# B&R Automation Studio project PLC code - cp (part 2)

### SM_i.ax
```
InitParameter (Version=5.02.1, NcSwId=ACP10)
  ACP10AXIS_typ:
    dig_in:
      level:
        reference = ncACTIV_HI
        pos_hw_end = ncACTIV_HI
        neg_hw_end = ncACTIV_HI
        trigger1 = ncACTIV_HI
        trigger2 = ncACTIV_HI
    encoder_if:
      parameter:
        count_dir = ncINVERSE
        scaling:
          load:
            units = 1000
            rev_motor = 1
    limit:
      parameter:
        v_pos = 10000.0
        v_neg = 10000.0
        a1_pos = 5000.0
        a2_pos = 5000.0
        a1_neg = 5000.0
        a2_neg = 5000.0
        t_jolt = 0.0
        t_in_pos = 0.0
        pos_sw_end = 2000000000
        neg_sw_end = -2000000000
        ds_warning = 100000.0
        ds_stop = 100000.0
        a_stop = 500000.0
        dv_stop = 0.0
        dv_stop_mode = ncOFF
    controller:
      mode = ncPOSITION
      position:
        kv = 50.0
        tn = 0.0
        t_predict = 0.02
        t_total = 0.02
        p_max = 1.0E+30
        i_max = 0.0
      speed:
        kv = 2.0
        tn = 0.0
        t_filter = 0.0
        isq_filter1:
          type = ncOFF
          a0 = 0.0
          a1 = 0.0
          b0 = 0.0
          b1 = 0.0
          b2 = 0.0
          c0_par_id = 0
          c1_par_id = 0
        isq_filter2:
          type = ncOFF
          a0 = 0.0
          a1 = 0.0
          b0 = 0.0
          b1 = 0.0
          b2 = 0.0
          c0_par_id = 0
          c1_par_id = 0
        isq_filter3:
          type = ncOFF
          a0 = 0.0
          a1 = 0.0
          b0 = 0.0
          b1 = 0.0
          b2 = 0.0
          c0_par_id = 0
          c1_par_id = 0
      uf:
        type = ncLINEAR
        auto_config = ncMOTOR_PAR
        u0 = 0.0
        un = 0.0
        fn = 50.0
        k_f_slip = 0.0
      ff:
        torque_load = 0.0
        torque_pos = 0.0
        torque_neg = 0.0
        kv_torque = 0.0
        inertia = 0.0
        t_filter_a = 0.0
    move:
      stop:
        parameter[0]:
          decel_ramp = ncA_LIMIT
          controller = ncON
        parameter[1]:
          decel_ramp = ncA_LIMIT
          controller = ncON
        parameter[2]:
          decel_ramp = ncA_LIMIT
          controller = ncON
        parameter[3]:
          decel_ramp = ncA_LIMIT
          controller = ncON
        quickstop:
          decel_ramp = ncA_LIMIT
          t_jolt = 0
        drive_error:
          decel_ramp = ncA_LIMIT
      homing:
        parameter:
          s = 0
          v_switch = 4000.0
          v_trigger = 4000.0
          a = 2000.0
          mode = ncDIRECT
          edge_sw = ncPOSITIVE
          start_dir = ncPOSITIVE
          trigg_dir = ncPOSITIVE
          ref_pulse = ncOFF
          fix_dir = ncOFF
          tr_s_block = 0.0
          torque_lim = 0.0
          ds_block = 0.0
          ds_stop = 0.0
      basis:
        parameter:
          v_pos = 2000.0
          v_neg = 2000.0
          a1_pos = 1000.0
          a2_pos = 1000.0
          a1_neg = 1000.0
          a2_neg = 1000.0
    message:
      text:
        parameter:
          format = ncBREAK
          columns = 80
          data_modul = acp10etxen
```

### DryerComms.var
```iecst
VAR
	gDryerLocalParams : Dryer_SwParameters; (*Local parameters*)
	gDryerLocalSignals : DryerRemoteData;
END_VAR
```

- RunTextScript.bat (not shown)

### ReadmePrinterConfigurator.txt
```
	From efi Cretaprint Almazora Castellon

(*
View of the machine from the Operator side

>>>>>> LeftHandMachine 					RightHandMachine <<<<<<<<
(BK_A #1 >> BK_B #2)		LOGICAL			(BK_A #2 << BK_B #1)

Vertical:	#2 									Vertical:	#3
IclaNode: 	#5									IclaNode: 	#7
IclaIndex:	#1									IclaIndex:	#2

	          ################-################
	          ################-################
	          ################-################
	          ################-################
	##########################-###########################
	##########################-###########################
	    ######################-#######################
	    ######################-#######################
	    ######################-#######################
	    ######################-#######################

	BLOCK A [1-physical]				BLOCK B [2-physical]

*)
```

### Program Logical/Dryer/Config/Initialize

#### Initialize.st
```iecst
PROGRAM _INIT

	HWInfoCpu.pName := ADR(gDryer.St.HwData.Name);
	HWInfoCpu.first := TRUE;
	HWInfoCpu.enable := TRUE;
	HWInfoCpu();
	gDryer.St.HwData.Family := HWInfoCpu.family;

	// Tranfer permanent vars when PLC is starting
	gMachine.St.HwData.SerialNumber := gPermanentSN;

	gDryer.Pt:= gPermanentDryer;
	gBelt.parSw := gPermanentSwBelt;
	gSimpleBlock[1].parSw := gPermanentSimpleBlock;
	gTransVacuum[1].parSw := gPermanentTrVacuum[1];
	gTransVacuum[2].parSw := gPermanentTrVacuum[2];
	gNirAdphos.Parameters := gPermanentNirAdphos;
	gArcLampGew.Parameters := gPermanentArcLampGew;

	gSimMachine.Parameters.MachineType := gPermanentSimMachinePar.MachineType;

END_PROGRAM

PROGRAM _CYCLIC

	//Assign the ConfigurationID been executed
	projectInfo(Execute:=gDryer.Pt.ConfigNameID=0); //Just to execute if still the configuration has not been read
	IF projectInfo.Done AND NOT projectInfo.Error THEN
		IF brsstrcmp(ADR(GC_CONFIG_DRYER_NOZ2),ADR(projectInfo.ConfigurationID))=0 THEN
			gDryer.Pt.ConfigNameID:=GC_CONFIG_DRYER_NOZ2_ID;
			gSimMachine.Parameters.MachineType := SIM_MACHINE_REAL;
		ELSIF brsstrcmp(ADR(GC_CONFIG_SIMDRYER_NOZ2),ADR(projectInfo.ConfigurationID))=0 THEN
			gDryer.Pt.ConfigNameID:=GC_CONFIG_SIMDRYER_NOZ2_ID;
		ELSE
			gDryer.Pt.ConfigNameID:=0;
		END_IF
		strcpy(ADR(gDryer.Pt.ConfigName),ADR(projectInfo.ConfigurationID));
	END_IF

END_PROGRAM
```

### Program Logical/Dryer/Config/MachineConfigurator

#### AsignCommonData.st
```iecst
ACTION AsignCommonData:

	//Just writing the fixed configuration once per each 5s
	IF NOT (EDGEPOS(gPLC.xBlk_5s) OR gPLC.xFirst_Scan OR xChangedSimMachine) THEN
		RETURN;
	END_IF

	////////////////////////////////////////////////////////////
	/////GENERAL	GENERAL		GENERAL		GENERAL	////////////
	////////////////////////////////////////////////////////////

	gDryer.Pt.CT.rMaxMargin		:= 25.0;
	gDryer.Pt.CT.rMinMargin		:= 5.0;
	gDryer.Pt.CT.rMinThicknessMedia		:= 1.0;
	gDryer.Pt.CT.rMaxThicknessMedia		:= 12.0;
	gDryer.Pt.CT.rDistanceThicknesToPD	:= 187.0;

	/////////////////////////////////////////////////////
	/////BELT	BELT	BELT	BELT	BELT	BELT/////
	/////////////////////////////////////////////////////

	gBelt.parameters.IndexAxis:=1;
	gBelt.parameters.rAcceleration := 1050;
	gBelt.parameters.rSoftDeceleration := 1000;
	gBelt.parameters.rDeceleration := 2200;
	gBelt.parameters.rMaxAcceleration := 1500.0;
	gBelt.parameters.rMaxDeceleration := 2500.0;
	gBelt.parameters.rMaxSpeed := gBelt.states.Hw.rMaxSpeed;

	// From Units measure to meters per minute
	gBelt.parameters.DriveUnit.TransmissionType := TRANS_LINEAL_PERIMETER;
	gBelt.parameters.DriveUnit.LinealPerimeter.PulsesPerTurn := GC_UNITS_BY_REV_DRIVE;
	gBelt.parameters.DriveUnit.LinealPerimeter.GearBox := gBelt.parSw.rGearBox;
	gBelt.parameters.DriveUnit.LinealPerimeter.Perimeter := gBelt.parSw.rAxisLength;

	gBelt.parameters.xExistBelt := TRUE;

	////////////////////////////////////////////////////////////////////////////////////////////////////////////
	// TRANSPORT VACUUM
	////////////////////////////////////////////////////////////////////////////////////////////////////////////
	FOR iIndexTrVacc := 1 TO MAX_LAST_TRANS_VACUUM DO
		gTransVacuum[iIndexTrVacc].Parameters.xInstalled := iIndexTrVacc <= gDryer.Pt.CT.iNumTransVacuum;

		gTransVacuum[iIndexTrVacc].Parameters.parPID.rKp := 0.4;
		gTransVacuum[iIndexTrVacc].Parameters.parPID.rTi := 1.5;
		gTransVacuum[iIndexTrVacc].Parameters.parPID.rKd := 0.0;
		gTransVacuum[iIndexTrVacc].Parameters.parPID.rTd := 0.0;

		gTransVacuum[iIndexTrVacc].Parameters.rMaxSystemVacuum := 18.0;
		gTransVacuum[iIndexTrVacc].Parameters.rMaxSpeed := 3000;
		IF gTransVacuum[iIndexTrVacc].Parameters.rMaxPIDOut = 0 THEN
			gTransVacuum[iIndexTrVacc].Parameters.rMaxPIDOut := 55.0;
		END_IF
	END_FOR
	/////////////////////////////////////////////////////
	/////MODEL	MODEL	MODEL	MODEL	MODEL	MODEL////
	/////////////////////////////////////////////////////

	gThicknessCtrl.parameters.sections[1].xEnabled := TRUE;
	gThicknessCtrl.parameters.iSections := 1;

	gThicknessCtrl.parameters.Detection.ProductDetect.pMediaInProductDetectL1 := gDryer.In.ProductDetect.pPDSignalSensorL1;
	gThicknessCtrl.parameters.Detection.ProductDetect.pMediaInProductDetectL2 := gDryer.In.ProductDetect.pPDSignalSensorL2;

	gThicknessCtrl.parameters.rMountedMediaHeigh := 75.0;

	gThicknessCtrl.parameters.pExtContMedia := ADR(gDryer.Pt.SW.Media);

	// JAM DETECTION DEVICES
	gDryer.Pt.CT.iNumSensorsPerJamDevice := 4;

END_ACTION
```

#### AsignDataDryerNoz2.st
```iecst
ACTION AsignDataDryerNoz2:

	//Just writing the fixed configuration once per each 5s
	IF NOT (EDGEPOS(gPLC.xBlk_5s) OR gPLC.xFirst_Scan OR xChangedSimMachine) THEN
		RETURN;
	END_IF

	////////////////////////////////////////////////////////////
	/////GENERAL	GENERAL		GENERAL		GENERAL	////////////
	////////////////////////////////////////////////////////////
	gDryer.Pt.CT.rMountedMediaLevelInBypassMode	:= 145.0;
	gDryer.Pt.CT.rMaxBeltTorque 		:= 25.0;
	gDryer.Pt.CT.rMaxBeltTempFast 		:= 190.0;
	gDryer.Pt.CT.rMaxBeltTempSlow 		:= 180.0;
	gDryer.Pt.SW.Safety.rMaxBeltSpeedSetPoint := 100.0;
	gDryer.Pt.PDSignalTpe 				:= PDCFG_CARRIAGE;
	gDryer.St.iJamDevices				:= 1;

	gBelt.parameters.xDriveProtectionOK := TRUE; //This machine doesn't have this signal connected to the PLC

	//Here are configured blocks in function of the machine direction
	//When machine is block then we need use correction as block physical 2 because PD is at the same distance than Block 1, for that is change process in function of machine 2 Blcoks or machine 1 block
	gSimpleBlock[1].parameters.iMotorAxisIndex := 2;

	////////////////////////////////////////////////////////////
	/////BLOCK	BLOCK	BLOCK	BLOCK	BLOCK	BLOCK///////////
	////////////////////////////////////////////////////////////
	FOR iIndexBlock:=1 TO gDryer.Pt.CT.iNumBlocks DO

		gSimpleBlock[iIndexBlock].In.xDifferentialOK := TRUE;
		gSimpleBlock[iIndexBlock].In.xDriveProtectionOK := TRUE;
		gSimpleBlock[iIndexBlock].In.xSafetyOK := TRUE;

		gSimpleBlock[iIndexBlock].parameters.Hw.xExistBlock := gDryer.Pt.MachineModel = DryerType_NOZ2_NIR_ARCLAMP;

		gSimpleBlock[iIndexBlock].parSw.xEnableToMovements := TRUE;
		gSimpleBlock[iIndexBlock].parSw.xEnableToPrint := TRUE;

		gSimpleBlock[iIndexBlock].parameters.Motor.rDriveManSpeed		:=10.0;
		gSimpleBlock[iIndexBlock].parameters.Motor.rDriveAutoSpeed		:=30.0;
		gSimpleBlock[iIndexBlock].parameters.Motor.rMinThicknessMedia:= gDryer.Pt.CT.rMinThicknessMedia;
		gSimpleBlock[iIndexBlock].parameters.Motor.rReduceSpeedDistance :=6.0;
		gSimpleBlock[iIndexBlock].parameters.Motor.rAcceleration		:= 172.5;
		gSimpleBlock[iIndexBlock].parameters.Motor.rDeceleration		:= 172.5;

		//Position parameters (mm)
		gSimpleBlock[iIndexBlock].parameters.Motor.rSafePosition	:= 85.0;//Max heigh (theoretically 100)
		gSimpleBlock[iIndexBlock].parameters.Motor.rMinSafePosition	:= 10.0;	//Min heigh
		gSimpleBlock[iIndexBlock].parameters.Motor.rCapPosition		:= 80.0;//CAP

		gSimpleBlock[iIndexBlock].parameters.Motor.DriveUnit.TransmissionType := TRANS_SCREW_PITCH;
		gSimpleBlock[iIndexBlock].parameters.Motor.DriveUnit.ScrewPitch.PulsesPerTurn := GC_UNITS_BY_REV_DRIVE;
		gSimpleBlock[iIndexBlock].parameters.Motor.DriveUnit.ScrewPitch.GearBox := 7.25;
		gSimpleBlock[iIndexBlock].parameters.Motor.DriveUnit.ScrewPitch.Pitch := 5.0;

		gSimpleBlock[iIndexBlock].parameters.Motor.rReferencePosition		:= 20.0;

		//Current Parameters
		gSimpleBlock[iIndexBlock].parameters.Motor.uiMaxCurrentBarsUp		:= 3;
		gSimpleBlock[iIndexBlock].parameters.Motor.uiMaxCurrentBarsDown		:= 1;

		gSimpleBlock[iIndexBlock].parameters.Motor.VerticalDirection:= MOTOR_POSITIVE;

	END_FOR

	///////////////////////////////////////////////////
	/////DING		DING		DING		DING  /////
	///////////////////////////////////////////////////
	gDing.Parameters.xDingInstalled := FALSE;

	///////////////////////////////////////////////////
	//////// DETECTION  DETECTION  DETECTION  /////////
	///////////////////////////////////////////////////

	gBasicDetectMedia.Parameters.xInstalled := TRUE;
	gBasicDetectMedia.Parameters.rCorrection := 12;

	/////////////////////////////////////////////////////
	/////   TRANSPORT_VACUUM  TRANSPORT_VACUUM   ////////
	/////////////////////////////////////////////////////
	gTransVacuum[1].Parameters.xInstalled := TRUE;
	gTransVacuum[1].Parameters.Hw.xSystemWithJoints := FALSE;
	gTransVacuum[1].Parameters.Hw.uiNumBlowers := 2;
	gTransVacuum[1].Parameters.Hw.BlowerData[1].iIndex := 1;
	gTransVacuum[1].Parameters.Hw.BlowerData[1].Direction := MOTOR_NEGATIVE;
	gTransVacuum[1].Parameters.Hw.BlowerData[2].iIndex := 2;
	gTransVacuum[1].Parameters.Hw.BlowerData[2].Direction := MOTOR_NEGATIVE;
	gTransVacuum[1].Parameters.xStartUpEnable := FALSE;
	gAxisInverter[gTransVacuum[1].Parameters.Hw.BlowerData[1].iIndex].Parameters.Hardware.CpuFamily := gDryer.St.HwData.Family;
	gAxisInverter[gTransVacuum[1].Parameters.Hw.BlowerData[2].iIndex].Parameters.Hardware.CpuFamily := gDryer.St.HwData.Family;

	/////////////////////////////////////////////////////
	///// ARCLAMP ARCLAMP ARCLAMP ARCLAMP ARCLAMP ///////
	/////////////////////////////////////////////////////

	gArcLampGew.Parameters.xInstalled := gDryer.Pt.MachineModel = DryerType_NOZ2_NIR_ARCLAMP;

	gArcLampGew.Parameters.CpuFamily := gDryer.St.HwData.Family;
	gArcLampGew.Parameters.iLampQuantity := 2;

	//With real machine, communications cannot be disabled
	IF gDryer.Pt.ConfigNameID <> GC_CONFIG_SIMDRYER_NOZ2_ID THEN
		gArcLampGew.Parameters.xDisableComms := FALSE;
	END_IF

	/////////////////////////////////////////////////////
	///// NIR NIR NIR NIR NIR NIR NIR NIR NIR NIR ///////
	/////////////////////////////////////////////////////
	gNirAdphos.Parameters.xInstalled := gDryer.Pt.MachineModel <> DryerNoType;

	gNirAdphos.Parameters.iTotalModules := 2;
	gNirAdphos.Parameters.CpuFamily := gDryer.St.HwData.Family;
	gNirAdphos.Parameters.rMaxSurfaceTemp := 50;

	gNirAdphos.Parameters.DDC.iLamps := 48;
	gNirAdphos.Parameters.DDC.pIntensityNir1 := ADR(gThicknessCtrl.status.Dry[1].Intensity);
	gNirAdphos.Parameters.DDC.pIntensityNir2 := ADR(gThicknessCtrl.status.Dry[2].Intensity);
	gNirAdphos.Parameters.DDC.rMinIntensityPercentage := 8.0;

	// Thermal inertia configuration
	// Assigning data just if no data to allow setting the data during research
	IF gDryer.Pt.ThermalInertia.iBoardsToStartReducing = 0 THEN
		gDryer.Pt.ThermalInertia.iBoardsToStartReducing := 60;
	END_IF
	IF gDryer.Pt.ThermalInertia.iBoardsToMaxPowerReduction = 0 THEN
		gDryer.Pt.ThermalInertia.iBoardsToMaxPowerReduction := 90;
	END_IF
	IF gDryer.Pt.ThermalInertia.rMaxPowerReduction = 0 THEN
		gDryer.Pt.ThermalInertia.rMaxPowerReduction := 0.85;
	END_IF

	/////////////////////////////////////////////////////
	/////MODEL	MODEL	MODEL	MODEL	MODEL	MODEL////
	/////////////////////////////////////////////////////

	//Configuring machine transport because some values are different in two blocks
	CASE gDryer.Pt.MachineModel OF
		DryerType_NOZ2_NIR,
		DryerType_NOZ2_NIR_ARCLAMP:
			gThicknessCtrl.parameters.iTotalBlocksLengh := 625;
			gThicknessCtrl.parameters.Belt.iDistanceEmptyBeltIni := 685;
	END_CASE;

	gThicknessCtrl.parameters.sections[1].xEnabled	:= TRUE;
	gThicknessCtrl.parameters.sections[1].iStart	:= 1;
	gThicknessCtrl.parameters.sections[1].iEnd		:= 250;

	gThicknessCtrl.parameters.Detection.Basic.xLoadMedia := TRUE;
	gThicknessCtrl.parameters.Detection.Basic.xEnableMediaTracking := TRUE;
	gThicknessCtrl.parameters.Detection.Basic.iMediaFilter := 1; // To avoid adding a 0 in the Tail section

	gThicknessCtrl.parameters.Dry.xEnableMediaTracking := TRUE;

	gThicknessCtrl.parameters.Dry.iLamps := 48;
	gThicknessCtrl.parameters.Dry.rLampOffset := -1435/2;
	gThicknessCtrl.parameters.Dry.rLampWidth := 1435.0/48.0;
	IF gThicknessCtrl.parameters.Dry.rThermalDelay = 0 THEN
		gThicknessCtrl.parameters.Dry.rThermalDelay := 500;
		gThicknessCtrl.parameters.Dry.rCommsDelay := 200;
	END_IF

	gThicknessCtrl.parameters.Dry.Dryers[1].iPosition := 290;
	gThicknessCtrl.parameters.Dry.Dryers[2].iPosition := 415;

	//gThicknessCtrl.parameters.CheckMedia[1].xActive := FALSE; // Deactivated due to sensor reading problems till new sensors will be implemented NOZDRYER-450
	gThicknessCtrl.parameters.CheckMedia[1].CheckPosition := 578;
	gThicknessCtrl.parameters.CheckMedia[1].CheckDelayPosition := 15;
	gThicknessCtrl.parameters.CheckMedia[2].CheckPosition := 578;
	gThicknessCtrl.parameters.CheckMedia[2].CheckDelayPosition := 15;
	gThicknessCtrl.parameters.CheckMedia[2].xActive := gDryer.Pt.SW.xDoubleLine;

	//Jam
	gJamDetect[1].Parameters.iSensorsQuantity := gDryer.Pt.CT.iNumSensorsPerJamDevice;
	gJamDetect[1].Parameters.xJamEnabled	:= TRUE;
	//There are no bars in the dryer, but to use this jam package, designed to be used one jam sensor per bar, we active 4 bars because we have 4 sensors. 2 per NIR module
	gJamDetect[1].Parameters.xBarInstalled[1]:= gNirAdphos.Parameters.xInstalled;
	gJamDetect[1].Parameters.xBarInstalled[2]:= gNirAdphos.Parameters.xInstalled;
	gJamDetect[1].Parameters.xBarInstalled[3]:= gNirAdphos.Parameters.xInstalled;
	gJamDetect[1].Parameters.xBarInstalled[4]:= gNirAdphos.Parameters.xInstalled;
	gJamDetect[1].Parameters.iLowJamCheckDuration[0] := T#1m;
	gJamDetect[1].Parameters.iLowJamTimes[0] := 3;
	gJamDetect[1].Parameters.iLowJamCheckDuration[1] := T#30m;
	gJamDetect[1].Parameters.iLowJamTimes[1] := 10;

END_ACTION
```

#### MachineConfigurator.st
```iecst
PROGRAM _INIT

	//Default values
	gDryerLocalParams.Media.rThickness := 2;
	gDryerLocalParams.Media.rMargin 	:= 10;
	gDryerLocalParams.Media.rLength := 1500;
	gDryerLocalParams.Media.rWidth := 600;

	gThicknessCtrl.parameters.CheckMedia[1].xActive := TRUE;

	//By default, working with comms simulation
	gArcLampGew.Parameters.xDisableComms := TRUE;

END_PROGRAM

PROGRAM _CYCLIC

	//Determine number of last block
	CASE gDryer.Pt.MachineModel OF

		DryerType_NOZ2_NIR,
		DryerType_NOZ2_NIR_ARCLAMP:
			gDryer.Pt.CT.iNumBlocks:=1;
			gDryer.Pt.CT.iNumTransVacuum := 1;
			gDryer.Pt.SW.xMachineDirection := 1; //Machine from left

	END_CASE;

	//Determine machine direction
	// RIGHT: gDryer.Pt.SW.xMachineDirection is 0 or FALSE
	// LEFT:  gDryer.Pt.SW.xMachineDirection is 1 or TRUE
	gDryer.Pt.xLeftHandMachine := gDryer.Pt.SW.xMachineDirection;
	gDryer.Pt.xRightHandMachine:= NOT gDryer.Pt.xLeftHandMachine;

	////////////////////////////////////////////////////////////////////////////////////////////////////////////
	// GENERAL
	////////////////////////////////////////////////////////////////////////////////////////////////////////////

	MachineModel;

	AsignCommonData;

	CASE gDryer.Pt.ConfigNameID OF

		GC_CONFIG_DRYER_NOZ2_ID:
			CASE gDryer.Pt.MachineModel OF
				DryerType_NOZ2_NIR,
				DryerType_NOZ2_NIR_ARCLAMP:
					AsignDataDryerNoz2;
			END_CASE

		GC_CONFIG_SIMDRYER_NOZ2_ID:
			CASE gSimMachine.Parameters.DryerType OF
				SIM_DRYER_NOZ2_NIR,
				SIM_DRYER_NOZ2_NIR_ARCLAMP:
					AsignDataDryerNoz2;
			END_CASE
	END_CASE

	DryerModelCopy := gDryer.Pt.MachineModel;

END_PROGRAM
```

### Program Logical/Dryer/Config/SavePermanent

#### SavePermanent.st
```iecst
PROGRAM _CYCLIC

	// Permanents Vars
	IF brsstrlen(ADR(gDryer.St.HwData.SerialNumber)) > 0 THEN
		gPermanentSN := gDryer.St.HwData.SerialNumber;
	END_IF
	gPermanentDryer:=gDryer.Pt;
	gPermanentSwBelt := gBelt.parSw;
	gPermanentSimpleBlock := gSimpleBlock[1].parSw;
	gPermanentTrVacuum[1] := gTransVacuum[1].parSw;
	gPermanentNirAdphos  := gNirAdphos.Parameters;
	gPermanentArcLampGew  := gArcLampGew.Parameters;

	gPermanentVersion.iVersion0 := gPLC.iVersion0;
	gPermanentVersion.iVersion1 := gPLC.iVersion1;
	gPermanentVersion.iVersion2 := gPLC.iVersion2;
	gPermanentVersion.iVersion3 := gPLC.iVersion3;

	gPermanentSimMachinePar:=gSimMachine.Parameters;

END_PROGRAM
```

### Program Logical/Dryer/DryerCtrl/DryerCtrl_Slow (IEC) - General program

#### Constants.var
```iecst
VAR CONSTANT
	BWMODE_OFF : UINT := 0; (*The blower never is turned on*)
	BWMODE_ON : UINT := 1; (*The blower always is turned on*)
	BWMODE_AUTO : UINT := 2; (*The blower is turned on while moving the belt and a configured time afterwards*)
	SHOT_MIN_TIME_BETWEEN_SHOTS : TIME := T#300MS; (*Minimum time between Printing Shots*)
	BEEP_START_COUNTS : USINT := 7;
END_VAR
```

#### AlarmsSlow.st
```iecst
ACTION AlarmsSlow:

	// Alarm: Platform Incoherence
	gDryer.Al.Alarm.xAlarmPlarformInc:= (gDryer.Pt.MachineModel=DryerNoType) AND NOT gDryer.St.Mode.xZero;

	gDryer.Al.Alarm.xNoActionDangerCollision := FALSE;

	// Warning: Max movemets because bent tile	// Warning: Max movemets because bent tile
	// Warning: Max movemets because bent tile	// Warning: Max movemets because bent tile
	IF EDGEPOS (gDryer.Al.Warning.xBentMedia) THEN
		iBentMediaCounter := iBentMediaCounter + 1;
	END_IF

	//If time without any change, decrease the count of movements
	tonDecreaseMovCount.IN := NOT gDryer.Al.Warning.xMaxMovsBentTile AND NOT gDryer.Al.Warning.xBentMedia AND NOT tonDecreaseMovCount.Q ;
	tonDecreaseMovCount.PT := T#5m;
	tonDecreaseMovCount();
	IF tonDecreaseMovCount.Q THEN
		//Safety decrease to avoid overflow
		iBentMediaCounter:= UINT_SUB(iBentMediaCounter,1);
	END_IF
	IF EDGEPOS(gDryer.Al.Warning.xMaxMovsBentTile) THEN
		iBentMediaCounter:= 0;
	END_IF

	IF 	iBentMediaCounter >= gc_diNumMaxManiobrasPDoblada THEN
		gDryer.Al.Warning.xMaxMovsBentTile:=TRUE;
	ELSIF  gDryer.AutoCmd.xReset THEN
		gDryer.Al.Warning.xMaxMovsBentTile:=FALSE;
	END_IF

	// Raising alarm of stopped media inside.
	// this is a simple way to reset the alarm. A more proper way to remove the alarm would be to
	// use a distanceVar in Thickness_Pos, but this is quite resource consuming, so this would be delayed
	IF gThicknessCtrl.status.MediaPosition.xMediaInside AND EDGENEG(gBelt.states.xRuningBelt) THEN
		gDryer.Al.Warning.xMediaStoppedInside := TRUE;
	ELSIF gThicknessCtrl.status.Belt.xBeltEmpty THEN
		gDryer.Al.Warning.xMediaStoppedInside := FALSE;
	END_IF

	//Sensors errors
	IF gDryer.In.Temp.xBeltSensorError THEN
		gDryer.Al.Warning.xBeltSensorError := TRUE;
	END_IF

	IF gDryer.In.Temp.xBoardInSensorError THEN
		gDryer.Al.Warning.xBoardInSensorError := TRUE;
	END_IF

	IF gDryer.In.Temp.xBoardOutSensorError THEN
		gDryer.Al.Warning.xBoardOutSensorError := TRUE;
	END_IF

	IF gDryer.In.Temp.xAirBlowerInputSensorError THEN
		gDryer.Al.Warning.xAirBlowerInputSensorError := TRUE;
	END_IF

	IF gDryer.In.Temp.xAirBlowerInputSensorError THEN
		gDryer.Al.Warning.xAirBlowerOutputSensorError := TRUE;
	END_IF

	//BELT ALARMS
	tonBeltOvertorque.IN := gBelt.states.rCurrentTorque > gDryer.Pt.CT.rMaxBeltTorque;
	tonBeltOvertorque.PT := t#120s;
	tonBeltOvertorque();
	IF tonBeltOvertorque.Q THEN
		gDryer.Al.Alarm.xAlrBeltOvertorque := TRUE;
	END_IF

	tonBeltOverTempFast.IN := gDryer.St.Temp.rBelt > gDryer.Pt.CT.rMaxBeltTempFast;
	tonBeltOverTempFast.PT := t#2s;
	tonBeltOverTempFast();
	IF tonBeltOverTempFast.Q THEN
		gDryer.Al.Alarm.xAlrBeltOverTempFast := TRUE;
	END_IF

	tonBeltOverTempSlow.IN := gDryer.St.Temp.rBelt > gDryer.Pt.CT.rMaxBeltTempSlow;
	tonBeltOverTempSlow.PT := t#30s;
	tonBeltOverTempSlow();
	IF tonBeltOverTempSlow.Q THEN
		gDryer.Al.Alarm.xAlrBeltOverTempSlow := TRUE;
	END_IF

	IF gJamDetect[1].Alarms.xAlrJamLowCrash THEN
		gDryer.Al.Warning.xJamLowCrash := TRUE;
	END_IF

	PsycallConfChecking;

END_ACTION

ACTION PsycallConfChecking:
	CASE gDryer.Pt.ConfigNameID OF
		GC_CONFIG_DRYER_NOZ2_ID:
			CASE gDryer.Pt.MachineModel OF
				DryerType_NOZ2_NIR,
				DryerType_NOZ2_NIR_ARCLAMP:
					plcCardsOK.0 := NOT X20DIF371_201.ModuleOk;
					plcCardsOK.1 := NOT X20DIF371_202.ModuleOk;
					plcCardsOK.2 := NOT X20DIF371_203.ModuleOk;
					//plcCardsOK.3 := NOT X20PS3300_204.ModuleOk;
					plcCardsOK.4 := NOT X20DOF322_205.ModuleOk;
					plcCardsOK.5 := NOT X20DOF322_206.ModuleOk;
					plcCardsOK.6 := NOT X20AI8321_207.ModuleOk;
					plcCardsOK.7 := NOT X20AO4622_208.ModuleOk;
					plcCardsOK.8 := NOT X20AT4222_209.ModuleOk;
					gDryer.Al.Alarm.xAlrWrongPhysConf := plcCardsOK>0;

				ELSE
					gDryer.Al.Alarm.xAlrWrongPhysConf := TRUE;
			END_CASE

		GC_CONFIG_SIMDRYER_NOZ2_ID:
			gDryer.Al.Alarm.xAlrWrongPhysConf := FALSE;

		ELSE

			gDryer.Al.Alarm.xAlrWrongPhysConf := TRUE;

	END_CASE

END_ACTION
```

#### CleanBelt.st
```iecst
ACTION CleanBelt:

	///////////////////////////////////////////////////////////////////////////////////////////////////////////////////
	// General conditions to clean belt	when machine is in AUTOMATIC OR MANUAL MODES
	///////////////////////////////////////////////////////////////////////////////////////////////////////////////////

	//Cleaning Belt by time. When cleaning, the time is reseted
	tonCleaningByTime.IN:= gBelt.states.xRuningBelt AND gDryer.Pt.SW.CleanBelt.xCleanBeltByTime AND NOT tonCleaningByTime.Q AND NOT xCleanBeltOrder;
	tonCleaningByTime.PT := MAX(tiCleaningBeltByTime, MIN_TIME_FOR_CLEANING_BELT); // Time converted from minutes to miliseconds
	tonCleaningByTime();

	//If the belt is not running, it is not possible to clean it
	IF NOT gBelt.states.xRuningBelt THEN
		RETURN;
	END_IF

	// Tiles counter
	IF gDryer.Pt.SW.CleanBelt.xCleanBeltByTiles AND (EDGEPOS (gDryer.St.xProductDetectL1) OR EDGEPOS(gDryer.St.xProductDetectL2)) THEN
		gDryer.Lg.iTilesCounterToClean:= gDryer.Lg.iTilesCounterToClean+1;
	END_IF

	//Cleaning by tiles. When cleaning, number of tiles is reseted
	IF gDryer.Pt.SW.CleanBelt.xCleanBeltByTiles AND (gDryer.Lg.iTilesCounterToClean >= INT_TO_UINT(iSPTilesToCleanBelt)) THEN
		xCleaningBeltByTiles:= TRUE;
	END_IF

	// Force cleaning applying delay. Why clean continuous is same that condition than force clean?
	IF gDryer.Pt.SW.CleanBelt.xCleanBeltForced THEN
		xCleanBeltForced:= TRUE;
		gDryer.Pt.SW.CleanBelt.xCleanBeltForced := FALSE;
	END_IF

	IF tonCleaningByTime.Q THEN
		xCleaningBeltByTime:=TRUE;
	END_IF

	IF xCleaningBeltByTiles OR xCleaningBeltByTime OR xCleanBeltForced OR gDryer.Pt.SW.CleanBelt.xCleanBeltContinue THEN
		xCleanBeltOrder:=TRUE;

		//Removed orders when cleaning
		xCleaningBeltByTiles:=FALSE;
		gDryer.Lg.iTilesCounterToClean:=0;
		xCleaningBeltByTime:=FALSE;
		xCleanBeltForced := FALSE;

	END_IF

	// Managing the duration of the belt cleaning
	tonCleaningBelt.IN:= xCleanBeltOrder;
	tonCleaningBelt.PT := MAX(gDryer.Pt.SW.CleanBelt.tiCleaningBeltDuration, MIN_DURATION_CLEANING_BELT);
	tonCleaningBelt();

	IF (tonCleaningBelt.Q AND NOT(gDryer.Pt.SW.CleanBelt.xCleanBeltContinue)) OR EDGENEG(gDryer.Pt.SW.CleanBelt.xCleanBeltContinue) THEN
		xCleanBeltOrder:=FALSE;
	END_IF

END_ACTION
```

#### GeneralMachineData.st
```iecst
ACTION GeneralMachineData:

	//////////////////////////////////////////////////////////////////////////////////////////////////////////////////////
	// BELT PARAMS      BELT PARAMS      BELT PARAMS      BELT PARAMS      BELT PARAMS      BELT PARAMS      BELT PARAMS
	// BELT PARAMS      BELT PARAMS      BELT PARAMS      BELT PARAMS      BELT PARAMS      BELT PARAMS      BELT PARAMS
	//////////////////////////////////////////////////////////////////////////////////////////////////////////////////////

	// Cleaning Belt limits cannot be lower than 1
	// Cleaning Belt parameters. Clean Belt disabled/enabled after delay
	tiCleaningBeltByTime	:= MINUTES_TO_TIME(gDryer.Pt.SW.CleanBelt.iCleaningBeltByTime);
	iSPTilesToCleanBelt		:= MAX (gDryer.Pt.SW.CleanBelt.iSPTilesToCleanBelt, MIN_TILES_FOR_CLEANING_BELT);

	////////// Belt Limits //////////////////////////////////
	//[RGP] Sending speed setpoint to gBelt. Not assigned directly from SW so maybe in the future SpeedSetpoint need to be used outside BeltPackage/BeltManager.
	//As done in previous lines by limiting maximum belt speed. //Not been able to have a Zero value in the SetPointSpeed
	gBelt.parameters.rSetPointSpeed := LIMIT(5.0, gDryer.Pt.SW.rBeltSpeedSetPoint, gDryer.Pt.SW.Safety.rMaxBeltSpeedSetPoint);

	// It gets belt direction following if machine configuration is left or right
	gBelt.parameters.Direction:= NOT gDryer.Pt.SW.xMachineDirection;

	////////////////////////////////////////////////////////////////////////////////////////////////////////////
	// MODEL
	////////////////////////////////////////////////////////////////////////////////////////////////////////////

	// Jetting Gap limits
	gDryer.Pt.SW.Media.rMargin:= LIMIT(gDryer.Pt.CT.rMinMargin,gDryer.Pt.SW.Media.rMargin,gDryer.Pt.CT.rMaxMargin);

	// Piece Tickness
	gDryer.Pt.SW.Media.rThickness:= LIMIT(gDryer.Pt.CT.rMinThicknessMedia,gDryer.Pt.SW.Media.rThickness,gDryer.Pt.CT.rMaxThicknessMedia);

	// Counters of shots printed by PD or by simulation
	//Counting out of any FOR. Makes no sense
	IF EDGEPOS (gDryer.St.xProductDetectL1) THEN
		gDryer.Lg.udiPiecesCounterL1:= gDryer.Lg.udiPiecesCounterL1+1;
	END_IF

	IF EDGEPOS (gDryer.St.xProductDetectL2) THEN
		gDryer.Lg.udiPiecesCounterL2:= gDryer.Lg.udiPiecesCounterL2+1;
	END_IF

	// Machine conversions
	gDryer.Lg.udiDifCounters:=0;

END_ACTION
```

#### SoundBeacon.st
```iecst
ACTION SoundBeacon:
	// Acoustic advise
	//
	// AutoReseteable Alarms sound management
	arFanBreakers		(xAlarm:= gDryer.Al.Alarm.xFanBreakers, xSilence:=gDryer.AutoCmd.xMuteAlarms);
	arFan24Vdc			(xAlarm:= gDryer.Al.Alarm.xFan24Vdc, xSilence:=gDryer.AutoCmd.xMuteAlarms);
	arMain24Vdc			(xAlarm:= gDryer.Al.Alarm.xMain24Vdc, xSilence:=gDryer.AutoCmd.xMuteAlarms);
	arBentMedia			(xAlarm:= gDryer.Al.Warning.xBentMedia, xSilence:=gDryer.AutoCmd.xMuteAlarms);
	arPDSensorErrorL1	(xAlarm:= gDryer.Al.Alarm.xPDBrokenSensorL1, xSilence:=gDryer.AutoCmd.xMuteAlarms);
	arPDSensorErrorL2	(xAlarm:= gDryer.Al.Alarm.xPDBrokenSensorL2, xSilence:=gDryer.AutoCmd.xMuteAlarms);
	arWrongPhysConf		(xAlarm:= gDryer.Al.Alarm.xAlrWrongPhysConf, xSilence:=gDryer.AutoCmd.xMuteAlarms);
	arAnyJam			(xAlarm:= gDryer.Al.Alarm.xAlrJam, xSilence:=gDryer.AutoCmd.xMuteAlarms);

	//arAnyStopAlarmMuted	(xAlarm:= gDryer.AlSummary.xAnyAlarm AND gDryer.St.StateMode<>PRINTERGEN_ZERO, xSilence:= gDryer.AutoCmd.xMuteAlarms);

	reasonSoundGen.1 := arFanBreakers.xAlarmSound;
	reasonSoundGen.2 := arFan24Vdc.xAlarmSound;
	reasonSoundGen.3 := arMain24Vdc.xAlarmSound;
	reasonSoundGen.4 := arBentMedia.xAlarmSound;
	reasonSoundGen.5 := arAnyStopAlarmMuted.xAlarmSound;
	reasonSoundGen.6 := arPDSensorErrorL1.xAlarmSound;
	reasonSoundGen.7 := arPDSensorErrorL2.xAlarmSound;
	reasonSoundGen.8 := arWrongPhysConf.xAlarmSound;
	reasonSoundGen.9 := arAnyJam.xAlarmSound;
	reasonSoundGen.25 := gBasicDetectMedia.AlSummary.xAlarmSound;
	reasonSoundGen.26 := gBelt.AlSummary.xAlarmSound;
	reasonSoundGen.27 := gSimpleBlock[1].AlSummary.xAlarmSound;
	reasonSoundGen.28 := gTransVacuum[1].AlSummary.xAlarmSound;
	reasonSoundGen.29 := gNirAdphos.AlSummary.xAlarmSound;
	reasonSoundGen.30 := gArcLampGew.AlSummary.xAlarmSound;
	reasonSoundGen.31 := gThicknessCtrl.Alarms.CheckMedia[1] OR gThicknessCtrl.Alarms.CheckMedia[2];

	gDryer.Al.xAlarmSound:= reasonSoundGen > 0;

	// Alarm sound output
	IF 	gDryer.AutoCmd.xMuteAlarms OR gDryer.In.Buttons.xZero THEN
		gDryer.AlSummary.xAlarmSound:=FALSE;
	ELSE
		gDryer.AlSummary.xAlarmSound:= gDryer.Al.xAlarmSound;
	END_IF;

	SoundAtStart;

	reasonBuzzer.0 := gDryer.AlSummary.xAlarmSound AND (iCountStartSound >= BEEP_START_COUNTS);
	reasonBuzzer.1 := gBelt.states.State = BELT_PREPARING_START  AND gPLC.xBlk_500ms;
	reasonBuzzer.2 := xStartSound;

	gDryer.Out.xBuzzer :=  reasonBuzzer > 0;

END_ACTION

ACTION SoundAtStart:

	//Whit 5, we have 3 beeps at the begining
	IF iCountStartSound >= BEEP_START_COUNTS THEN
		RETURN;
	END_IF

	tonStartSound.IN := NOT tonStartSound.Q;
	tonStartSound.PT := t#1s;
	tonStartSound();

	IF EDGEPOS(tonStartSound.Q) THEN
		iCountStartSound := iCountStartSound + 1;
	END_IF

	xStartSound := (iCountStartSound MOD 2) = 0;

END_ACTION
```

### Program Logical/Dryer/DryerCtrl/DryerCtrl_Fast (IEC) - Machine program

#### DryerCtrl_Fast.var
```iecst
VAR
	xRunBeltNormal : BOOL;
	xRunBeltLab : BOOL;
	xStopBeltWhileCleaning : BOOL;
	xSignalsStopBeltAuto : BOOL;
	xUserRaisesBlocks : BOOL;
	xOrdersRunBeltProduction : BOOL;
	xRunBeltByPass : BOOL;
	xAlarmsStopBeltRun : BOOL;
	enPrinterState : enumEFI_GenMachineState := PRINTERGEN_MANUAL; (*PRINTERGEN_ZERO*)
	enPrinterStatesInAuto : enumEFI_MachineState := PRINTERGEN_ZERO; (*PRINTERGEN_ZERO*)
	rsRunBeltOrderManual : RS;
	srPauseMachine : {REDUND_UNREPLICABLE} RS;
	stDryerAlarmsSummaryReseted : stEFI_AlarmSummary; (*stDingAlarmsReseted : stPhotoCellsAlarms;*)
	stDryerAlarmsReseted : Dryer_Alarms;
	tonStartButton : TON;
	ton_ZeroMode : TON;
	tpAlrBentMedia : TP;
	iIndexBlock : USINT;
	iReasonOut : UDINT;
	iReasonStopGen : UDINT;
	iReasonCritical : UDINT;
	stEventLogState : EventLog_typ;
	stEventLogOutAuto : EventLog_typ;
	stEventLog : EventLog_typ;
	stEventLogStopDrying : EventLog_typ;
	stEventLogCritical : EventLog_typ;
	g_xRunBeltOrderManual : BOOL; (*Belt order in manual filtered*)
	g_xRunBeltOrderAuto : BOOL; (*Belt order in auto*)
	reasonAnyWarningGen : UDINT;
	xEnabledAlarmPDSensor1 : BOOL;
	xEnabledAlarmPDSensor2 : BOOL;
	usiIndex : USINT;
	trgMountedTile : RF_TRIG;
	AutoLocationPrevious : MachineAutoLocation_enum;
	AutoLocationReseted : MachineAutoLocation_enum := MACHLOC_UNDEFINED;
	DryerCommandsReseted : {REDUND_UNREPLICABLE} Dryer_commands_Auto; (*Local parameters*)
	DryerSignalsAuto : REFERENCE TO DryerRemoteData; (*Local parameters*)
	DryerParams : REFERENCE TO Dryer_SwParameters; (*Local parameters*)
	iLastReasonStop : USINT;
	iReasonStop : USINT;
	iReasonSetPause : USINT;
	iReasonResetPause : USINT;
	DryerStatus : DryerMachineStatus_enum;
	DryerStatus_copy : DryerMachineStatus_enum;
	iReasonReadyToDry : USINT;
	xStartedAutoMan : BOOL;
	InputsSwReseted : Dryer_Inputs_Sw;
	tonMovingBeltAfterStop : TON;
END_VAR
VAR CONSTANT
	iHistoryLines : USINT := 25;
END_VAR
VAR
	StateHistory : ARRAY[0..iHistoryLines] OF DryerMachineStatus_enum;
	iIndexHistory : USINT;
	xNirReady : BOOL;
	xArcLampReady : BOOL;
	xAllDryersReady : BOOL;
	xNirStopped : BOOL;
	xArcLampStopped : BOOL;
	xAllDryersStopped : BOOL;
	xNirDrying : BOOL;
	xArcLampDrying : BOOL;
	xAllDryersDrying : BOOL;
	xChangeState : BOOL;
	iReasonSafetyEStop : UINT;
	tonStop : TON;
	xAnyDeviceEnabled : BOOL;
	iReasonJam : UINT;
	iReasonNotEnterAuto : UINT;
	xEdgeStop : BOOL;
	xOrderToCapReceived : BOOL;
	xOrderToPrintReceived : BOOL;
	iReasonCap : UINT;
	iReasonPrint : UINT;
	lastReasonCap : UINT;
	iBlockExecutionsOrder : UDINT;
	lastReasonPrint : UINT;
	iBlockDelay : UDINT;
	gDryerLocalSignalsReseted : DryerRemoteData;
	iReasonStopDrying : UINT;
	tonPreparingEmptyBelt : TON;
	iReasonKeepBlowersOn : UINT;
	xKeepBlowersOn : BOOL; (*To keep blowers running due to certain conditions*)
	xPDCarriageSignalL1 : REFERENCE TO BOOL; (*Use just in MachineInputs*)
	xPDCarriageSignalL2 : REFERENCE TO BOOL; (*Use just in MachineInputs*)
	ton_EmptyBelt : TON;
END_VAR
```

#### Alarms.st
```iecst
ACTION Alarms:

	// SAFETY
	IF NOT gDryer.In.Safety.xEStopFrontOK THEN gDryer.Al.Alarm.Safety.xEStopFront := TRUE; END_IF
	IF NOT gDryer.In.Safety.xEStopRearOK THEN gDryer.Al.Alarm.Safety.xEStopRear := TRUE; END_IF
	//IF NOT gDryer.In.Safety.xRemoteEStopOK THEN gDryer.Al.Alarm.Safety.xRemoteEStop := TRUE; END_IF  //TODO: Remove when working

	IF NOT gDryer.In.Safety.xMovementsEnabled THEN gDryer.Al.Warning.xNotEnabledMovement := TRUE; END_IF

	IF NOT gDryer.In.Safety.xClosedFrontInput OR NOT gDryer.In.Safety.xClosedFrontOutput THEN
		gDryer.Al.Warning.xFrontDoorOpened := TRUE;
	END_IF
	IF NOT gDryer.In.Safety.xClosedRearInput OR NOT gDryer.In.Safety.xClosedRearOutput THEN
		gDryer.Al.Warning.xRearDoorOpened := TRUE;
	END_IF

	iReasonSafetyEStop.0 := gDryer.Al.Alarm.Safety.xEStopFront;
	iReasonSafetyEStop.1 := gDryer.Al.Alarm.Safety.xEStopRear;
	iReasonSafetyEStop.2 := gDryer.Al.Alarm.Safety.xRemoteEStop;
	gDryer.Al.xAlrSafetySystemEStop := iReasonSafetyEStop>0;

	// Warning Alarm raised when a new BentTile is detected. The signal is kept for 5s
	tpAlrBentMedia.IN:=(gDryer.St.AutoMode.xProdORLab) AND EDGEPOS(gThicknessCtrl.status.Heigh.xIncreasedHeigh[1]);
	tpAlrBentMedia.PT:= T#5S;
	tpAlrBentMedia();
	gDryer.Al.Warning.xBentMedia:=tpAlrBentMedia.Q;

	//Count all the increase of heigh of the blocks as bent media
	IF EDGEPOS (tpAlrBentMedia.IN) THEN
		gDryer.Lg.udiBentTilesCounter:= gDryer.Lg.udiBentTilesCounter+1;
	END_IF

	//24VDC Power Supply for IDS
	IF NOT gDryer.In.xMain24VdcOK THEN gDryer.Al.Alarm.xMain24Vdc := TRUE; END_IF
	IF NOT gDryer.In.xFan24VdcOK THEN gDryer.Al.Alarm.xFan24Vdc := TRUE; END_IF
	IF NOT gDryer.In.xFanBreakersOK THEN gDryer.Al.Alarm.xFanBreakers := TRUE; END_IF
	IF gDryer.In.xFanBreakersWarning THEN gDryer.Al.Warning.xFanBreakersHighLoad := TRUE; END_IF

	// Alarm: xUpNotConsent
	gDryer.Al.Alarm.xUpNotConsent:= gDryer.St.AutoMode.xProduction AND
									NOT gDryer.St.xConsent;

	//Alarm: Mounted Piece Inide the Machine
	gDryer.Al.Alarm.xAlarmMountedMedia := gBasicDetectMedia.Alarms.xMountedMedia;
	gDryer.Al.Warning.xMountedMediaInside := gThicknessCtrl.status.MediaPosition.xMountedMediaInside;

	//Jam alarms
	iReasonJam.0 := gJamDetect[1].AlSummary.xAlarmStop;
	iReasonJam.1 := gArcLampGew.Alarms.xJam;
	iReasonJam.2 := gNirAdphos.Alarms.xAnyJam;
	iReasonJam.3 := gJamDetect[1].Alarms.xAlrJamCrash[1];
	iReasonJam.4 := gJamDetect[1].Alarms.xAlrJamCrash[2];
	iReasonJam.5 := gJamDetect[1].Alarms.xAlrJamCrash[3];
	iReasonJam.6 := gJamDetect[1].Alarms.xAlrJamCrash[4];
	//iReasonJam.7 := gThicknessCtrl.Alarms.CheckMedia[1] OR gThicknessCtrl.Alarms.CheckMedia[2];
	IF iReasonJam>0 THEN
		gDryer.Al.Alarm.xAlrJam := TRUE;
	END_IF

	IF gDryer.In.xOpenDoorsKey THEN
		gDryer.Al.Warning.xKeyMantenanceActive := TRUE;
	END_IF

	//Alarm: Broken PD
	CalcPDSensorAlarm;

END_ACTION

ACTION CalcPDSensorAlarm:

	//When no sensor is connected, cannot be checked
	IF (gDryer.Pt.PDSignalTpe <> PDCFG_SENSOR AND gDryer.Pt.PDSignalTpe <> PDCFG_SENSOR_AND_CARRIAGE) THEN
		gDryer.Lg.udiPiecesCounterErrorL1 := 0;
		gDryer.Lg.udiPiecesCounterErrorL2 := 0;
		RETURN;
	END_IF

	//Reset counter when belt is stoped or not in printin
	IF NOT gBelt.states.xRuningBelt OR NOT gDryer.St.Position.xInPrint THEN
		gDryer.Lg.udiPiecesCounterErrorL1 := 0;
		gDryer.Lg.udiPiecesCounterErrorL2 := 0;
		RETURN;
	END_IF

//	//Sensor 1
//	xEnabledAlarmPDSensor1 := NOT gDryer.Pt.SW.Dtp.xDoubleLine OR (gDryer.Pt.SW.Dtp.xDoubleLine AND gDryer.Pt.SW.Dtp.iModeLine1 = GC_DTP_RUN AND gDryer.Pt.SW.Dtp.iModeLine2 = GC_DTP_STOP);
//	T_AlarmPDL1.IN:= xEnabledAlarmPDSensor1 AND NOT gDryer.In.ProductDetect.xPDSignalSensorL1 AND gDryer.St.xMediaDetected;						//If Photocell1 Detect Tile and PD not
//	T_AlarmPDL1.PT:= REAL_TO_TIME( 60 * (gDryer.Pt.CT.rDistanceThicknesToPD + 8) / gBelt.states.rCurrentSpeed);		//In a time (depends of belt speed and distance between sensors). Adding 8mm safety
//	T_AlarmPDL1();
//	IF EDGEPOS(T_AlarmPDL1.Q) THEN gDryer.Lg.udiPiecesCounterErrorL1 := gDryer.Lg.udiPiecesCounterErrorL1 + 1; END_IF	//Increase Error Detect Counter
//
//	//Sensor 2
//	xEnabledAlarmPDSensor2 := gDryer.Pt.SW.Dtp.xDoubleLine AND gDryer.Pt.SW.Dtp.iModeLine1 = GC_DTP_STOP AND gDryer.Pt.SW.Dtp.iModeLine2 = GC_DTP_RUN;
//	T_AlarmPDL2.IN:= xEnabledAlarmPDSensor2 AND NOT gDryer.In.ProductDetect.xPDSignalSensorL2 AND gDryer.St.xMediaDetected;
//	T_AlarmPDL2.PT:= REAL_TO_TIME( 60 * (gDryer.Pt.CT.rDistanceThicknesToPD + 8) / gBelt.states.rCurrentSpeed);		//In a time (depends of belt speed and distance between sensors). Adding 8mm safety
//	T_AlarmPDL2();
//	IF EDGEPOS(T_AlarmPDL2.Q) THEN gDryer.Lg.udiPiecesCounterErrorL2 := gDryer.Lg.udiPiecesCounterErrorL2 + 1; END_IF

	IF gDryer.Lg.udiPiecesCounterErrorL1 > 10 THEN gDryer.Al.Alarm.xPDBrokenSensorL1:= TRUE; END_IF
	IF gDryer.Lg.udiPiecesCounterErrorL2 > 10 THEN gDryer.Al.Alarm.xPDBrokenSensorL2:= TRUE; END_IF

END_ACTION
```

#### AlarmsSummary.st
```iecst
ACTION AlarmsSummary:

	gDryer.Al.xAlrDisableGoToProduction := FALSE;

	// Safety alarms
	gDryer.AlSummary.xAlrSafetySystemGeneral:= gDryer.Al.xAlrSafetySystemEStop;

	//////////////////
	// General Summary
	//////////////////

	//Stop drying alarms
	iReasonStopDrying.0 := gDryer.Al.Alarm.xAlrBeltOvertorque;
	iReasonStopDrying.1 := gDryer.Al.Alarm.xAlrBeltOverTempFast;
	iReasonStopDrying.2 := gDryer.Al.Alarm.xAlrBeltOverTempSlow;

	gDryer.Al.xAlrStopDrying :=  iReasonStopDrying > 0;
	//Register the reason of the Critical Alarm
	IF gDryer.St.Mode.xAuto AND EDGEPOS(gDryer.Al.xAlrStopDrying) THEN
		gDryer.Al.iReasonStopDrying := iReasonStopDrying;
		LogStopDryingAlarm;
	ELSIF EDGEPOS(gDryer.St.Mode.xAuto AND NOT gDryer.Al.xAlrStopDrying) THEN
		gDryer.Al.iReasonStopDrying := 0;
	END_IF

	//Warnings//
	reasonAnyWarningGen.0 := gDryer.Al.Alarm.xAlarmPlarformInc;
	reasonAnyWarningGen.1 := gDryer.Al.Alarm.xNoActionDangerCollision;
	reasonAnyWarningGen.2 := gDryer.Al.Warning.xBentMedia;
	reasonAnyWarningGen.3 := gDryer.Al.Warning.xMaxMovsBentTile;
	reasonAnyWarningGen.4 := gDryer.Al.Warning.xValidConfiguration;
	reasonAnyWarningGen.5 := gBelt.AlSummary.xAnyWarning;
	reasonAnyWarningGen.6 := gDryer.Al.Warning.xAirBlowerInputSensorError;
	reasonAnyWarningGen.7 := gDryer.Al.Warning.xAirBlowerOutputSensorError;
	reasonAnyWarningGen.8 := gDryer.Al.Warning.xBeltSensorError;
	reasonAnyWarningGen.9 := gDryer.Al.Warning.xBoardInSensorError;
	reasonAnyWarningGen.10 := gDryer.Al.Warning.xBoardOutSensorError;
	reasonAnyWarningGen.11 := gDryer.Al.Warning.xFanBreakersHighLoad;
	reasonAnyWarningGen.12 := gDryer.Al.Warning.xFrontDoorOpened;
	reasonAnyWarningGen.13 := gDryer.Al.Warning.xRearDoorOpened;
	reasonAnyWarningGen.14 := gDryer.Al.Warning.xKeyMantenanceActive;
	reasonAnyWarningGen.15 := gDryer.Al.Warning.xMediaStoppedInside;
	reasonAnyWarningGen.16 := gDryer.Al.Warning.xMountedMediaInside;
	reasonAnyWarningGen.17 := gDryer.Al.Warning.xJamLowCrash;

	gDryer.AlSummary.xAnyWarning:= reasonAnyWarningGen>0;

	//Any ALarm//
	gDryer.AlSummary.xAnyAlarm:= gDryer.AlSummary.xAlarmCritical OR gDryer.AlSummary.xAlarmStop;

	//Critial alarms//
	iReasonCritical.0 := gDryer.AlSummary.xAlrSafetySystemGeneral;
	iReasonCritical.1 := gBelt.AlSummary.xAlarmCritical;
	iReasonCritical.2 := gNirAdphos.AlSummary.xAlarmCritical;
	iReasonCritical.3 := gArcLampGew.AlSummary.xAlarmCritical;
	iReasonCritical.4 := gTransVacuum[1].AlSummary.xAlarmCritical;

	gDryer.AlSummary.xAlarmCritical:=  iReasonCritical > 0;
	//Register the reason of the Critical Alarm
	IF gDryer.St.Mode.xAuto AND EDGEPOS(gDryer.AlSummary.xAlarmCritical) THEN
		gDryer.AlSummary.iReasonCritical := iReasonCritical;
		LogCriticalAlarm;
	ELSIF EDGEPOS(gDryer.St.Mode.xAuto AND NOT gDryer.AlSummary.xAlarmCritical) THEN
		gDryer.AlSummary.iReasonCritical := 0;
	END_IF

	//Alarms stop//
	iReasonStopGen.0 := gDryer.Al.Alarm.xMain24Vdc;
	iReasonStopGen.1 := gDryer.Al.Alarm.xAlarmComPcPLC;
	iReasonStopGen.2 := gDryer.Al.Alarm.xAlarmMountedMedia;
	iReasonStopGen.3 := gDryer.Al.Alarm.xAlrBeltOvertorque;
	iReasonStopGen.4 := gDryer.Al.Alarm.xAlrBeltOverTempFast;
	iReasonStopGen.5 := gDryer.Al.Alarm.xAlrBeltOverTempSlow;
	iReasonStopGen.6 := gBelt.AlSummary.xAlarmStop;
	iReasonStopGen.7 := gSimpleBlock[1].AlSummary.xAlarmStop;
	iReasonStopGen.8 := gNirAdphos.AlSummary.xAlarmStop;
	iReasonStopGen.9 := gArcLampGew.AlSummary.xAlarmStop;
	iReasonStopGen.10 := gTransVacuum[1].AlSummary.xAlarmStop;
	iReasonStopGen.11 := gNirAdphos.Alarms.xAnyJam; //Jam alarms always stop even not enabled
	iReasonStopGen.12 := gArcLampGew.Alarms.xJam; //Jam alarms always stop even not enabled
	iReasonStopGen.13 := gJamDetect[1].AlSummary.xAlarmStop;
	iReasonStopGen.14 := gThicknessCtrl.Alarms.CheckMedia[1] OR gThicknessCtrl.Alarms.CheckMedia[2];
	iReasonStopGen.15 := gDryer.Al.Alarm.xAlrJam;
	iReasonStopGen.16 := NOT gJamDetect[1].Inputs.xJamCrash[1] AND gBelt.states.xRuningBelt;
	iReasonStopGen.17 := NOT gJamDetect[1].Inputs.xJamCrash[2] AND gBelt.states.xRuningBelt;
	iReasonStopGen.18 := NOT gJamDetect[1].Inputs.xJamCrash[3] AND gBelt.states.xRuningBelt;
	iReasonStopGen.19 := NOT gJamDetect[1].Inputs.xJamCrash[4] AND gBelt.states.xRuningBelt;

	gDryer.AlSummary.xAlarmStop:= iReasonStopGen > 0;
	//Register the reason of the Alarm
	IF NOT gDryer.St.AutoMode.xStop AND EDGEPOS(gDryer.AlSummary.xAlarmStop) THEN
		gDryer.AlSummary.iReasonStop[0] := iReasonStopGen;
		LogStopAlarm;
	ELSIF EDGEPOS(NOT gDryer.St.AutoMode.xStop AND NOT gDryer.AlSummary.xAlarmStop) THEN
		gDryer.AlSummary.iReasonStop[0] := 0;
	END_IF

END_ACTION
```

#### AutoLocal.st
```iecst
ACTION AutoLocal:

	//This action just for Auto Local
	IF NOT gDryer.St.Mode.xAuto OR NOT gDryer.St.AutoLocation.xLocal THEN
		RETURN;
	END_IF

	IF EDGEPOS(gDryer.In.Sw.xStart_GI) THEN
		DryerSignalsAuto.Commands.xRunTransport := TRUE;
		DryerSignalsAuto.Commands.xPrepareToDry := TRUE;
		DryerSignalsAuto.Commands.xStartDrying := TRUE;
		xStartedAutoMan := TRUE;
	END_IF

	IF EDGEPOS(gDryer.In.Sw.xStop_GI) OR EDGEPOS(gDryer.In.Buttons.xStop) THEN
		DryerSignalsAuto.Commands.xPrepareToDry := FALSE;
		DryerSignalsAuto.Commands.xStartDrying := FALSE;
		xStartedAutoMan := FALSE;
	END_IF

	IF EDGEPOS(gDryer.In.Sw.xStop_GI) AND DryerStatus = DRYERMACH_MOVING THEN
		DryerSignalsAuto.Commands.xRunTransport := FALSE;
	END_IF

	tonMovingBeltAfterStop.IN := NOT xStartedAutoMan;
	tonMovingBeltAfterStop.PT := T#30s;
	tonMovingBeltAfterStop();

	IF tonMovingBeltAfterStop.Q AND gThicknessCtrl.status.Belt.xBeltEmpty THEN
		DryerSignalsAuto.Commands.xRunTransport := FALSE;
		gDryer.In.Sw.xStop_GI := TRUE;
	END_IF

END_ACTION
```

#### DryerCtrl_Fast.st
```iecst
PROGRAM _INIT
	//Avoid starting without an AutoLocation defined
	AutoLocationPrevious := MACHLOC_LOCAL;
END_PROGRAM

PROGRAM _CYCLIC

	//Inputs to the machine
	MachineInputs;

	// Reset general alarms
	IF gDryer.AutoCmd.xReset THEN

		//Enable resetting the alarm
		IF gDryer.Al.Alarm.xPDBrokenSensorL1 THEN
			gDryer.Lg.udiPiecesCounterErrorL1 := 0;
		END_IF
		IF gDryer.Al.Alarm.xPDBrokenSensorL2 THEN
			gDryer.Lg.udiPiecesCounterErrorL2 := 0;
		END_IF

		ResetAlarms;
	END_IF

	Alarms;
	AlarmsSummary;

	// ACTIONS
	MachineStates;

	DryerState;

	IF gDryer.St.AutoLocation.xLocal OR gDryer.St.AutoLocation.xLocalORManual THEN
		AutoLocal;
	END_IF

	// Update status and send more commands
	OrdersPrinter;

	//Reset Edge commands received from Sw
	gDryer.In.Sw := InputsSwReseted;

	gDryer.St.exec.fast := gDryer.St.exec.fast +1;

END_PROGRAM
```

#### DryerState.st
```iecst
ACTION DryerState:

	xAnyDeviceEnabled := gNirAdphos.Status.xEnabledNir OR gArcLampGew.Status.xEnabledArcLamp;
	xNirReady := gNirAdphos.State = NIRADPEW_READY OR gNirAdphos.State = NIRADPEW_RUNNING;
	xNirDrying := gNirAdphos.State = NIRADPEW_RUNNING;
	xNirStopped := gNirAdphos.State = NIRADPEW_IDLE OR gNirAdphos.State = NIRADPEW_ERROR;

	xArcLampReady := gArcLampGew.State = ARCLGEW_READY OR gArcLampGew.State = ARCLGEW_RUNNING;
	xArcLampDrying := gArcLampGew.State = ARCLGEW_RUNNING;
	xArcLampStopped := gArcLampGew.State = ARCLGEW_IDLE OR gArcLampGew.State = ARCLGEW_ERROR;

	xAllDryersReady := (xNirReady OR NOT gNirAdphos.Status.xEnabledNir) AND
						(xArcLampReady OR NOT gArcLampGew.Status.xEnabledArcLamp);
	xAllDryersDrying := (xNirDrying OR NOT gNirAdphos.Status.xEnabledNir) AND
						(xArcLampDrying OR NOT gArcLampGew.Status.xEnabledArcLamp);
	xAllDryersStopped := (xNirStopped OR NOT gNirAdphos.Status.xEnabledNir) AND
						(xArcLampStopped OR NOT gArcLampGew.Status.xEnabledArcLamp);

	tonPreparingEmptyBelt.IN := DryerStatus = DRYERMACH_PREPARINGEMPTYBELT AND gTransVacuum[1].Status.State <> TRANSVAC_OFF;
	tonPreparingEmptyBelt.PT := T#10s;
	tonPreparingEmptyBelt();

	CASE DryerStatus OF

		DRYERMACH_STOPPED:

			ResetOrdersToAllDryersDevices;

			IF DryerSignalsAuto.Commands.xRunTransport THEN
				DryerStatus:=DRYERMACH_PREPARINGTOMOVE;
			ELSIF DryerSignalsAuto.Commands.xPrepareToEmptyBelt THEN
				DryerStatus := DRYERMACH_PREPARINGEMPTYBELT;
			END_IF

		DRYERMACH_STOPPING_TRANSPORT:
			//Actions
			xOrdersRunBeltProduction := FALSE;
			gArcLampGew.Commands.xStop := TRUE;
			gNirAdphos.Commands.xStop := TRUE;

			//Transition
			IF NOT gBelt.states.xRuningBelt THEN
				DryerSignalsAuto.Commands := DryerCommandsReseted;
				DryerStatus:=DRYERMACH_STOPPED;
			END_IF

		DRYERMACH_PREPARINGEMPTYBELT:
			IF tonPreparingEmptyBelt.Q THEN
				gDryer.St.Out.xReadyToEmptyBelt := TRUE;
			END_IF
			IF DryerSignalsAuto.Commands.xRunTransport THEN
				DryerStatus := DRYERMACH_PREPARINGTOMOVE;
				gDryer.St.Out.xReadyToEmptyBelt := FALSE;
			END_IF

		DRYERMACH_PREPARINGTOMOVE:
			xOrdersRunBeltProduction := TRUE;

			IF gBelt.states.xRuningBelt THEN
				DryerStatus:=DRYERMACH_MOVING;
			END_IF

		DRYERMACH_MOVING:
			IF xAnyDeviceEnabled AND DryerSignalsAuto.Commands.xPrepareToDry THEN
				DryerStatus:=DRYERMACH_PREPARING;
			END_IF

		DRYERMACH_PREPARING:
			//Actions
			IF xChangeState THEN
				gArcLampGew.Commands.xPrepare := TRUE;
				gNirAdphos.Commands.xPrepare := TRUE;
			END_IF

			IF xAllDryersReady THEN
				DryerStatus:=DRYERMACH_PREPARED;
			END_IF

			IF NOT DryerSignalsAuto.Commands.xPrepareToDry THEN
				DryerStatus:=DRYERMACH_STOPPING_DRYING;
			END_IF

		DRYERMACH_PREPARED:
			IF DryerSignalsAuto.Commands.xStartDrying THEN
				DryerStatus:=DRYERMACH_STARTING;
			END_IF

			IF NOT DryerSignalsAuto.Commands.xPrepareToDry THEN
				DryerStatus:=DRYERMACH_STOPPING_DRYING;
			END_IF

		DRYERMACH_STARTING:
			//Actions
			IF xChangeState THEN
				gArcLampGew.Commands.xStart := TRUE;
				gNirAdphos.Commands.xStart := TRUE;
			END_IF

			//Transition
			IF xAllDryersDrying THEN
				DryerStatus:=DRYERMACH_DRYING;
			END_IF
			//Transition
			IF NOT DryerSignalsAuto.Commands.xStartDrying OR NOT DryerSignalsAuto.Commands.xPrepareToDry THEN
				DryerStatus:=DRYERMACH_STOPPING_DRYING;
			END_IF

		DRYERMACH_DRYING:
			IF NOT DryerSignalsAuto.Commands.xStartDrying OR gDryer.Al.xAlrStopDrying THEN
				DryerStatus:=DRYERMACH_STOPPING_DRYING;
			END_IF

		DRYERMACH_STOPPING_DRYING:
			//Actions
			IF xChangeState THEN
				gArcLampGew.Commands.xStop := TRUE;
				gNirAdphos.Commands.xStop := TRUE;
			END_IF

			IF xAllDryersStopped THEN
				DryerStatus:=DRYERMACH_MOVING;
			END_IF
			IF DryerSignalsAuto.Commands.xStartDrying THEN
				DryerStatus:=DRYERMACH_STARTING;
			END_IF

	END_CASE;

	IF (NOT gDryer.St.AutoMode.xProduction OR NOT DryerSignalsAuto.Commands.xRunTransport) AND DryerStatus<>DRYERMACH_STOPPED AND DryerStatus<>DRYERMACH_STOPPING_TRANSPORT AND DryerStatus<>DRYERMACH_PREPARINGEMPTYBELT THEN
		DryerStatus:=DRYERMACH_STOPPING_TRANSPORT;
	END_IF

	xChangeState := DryerStatus <> DryerStatus_copy;
	DryerStatus_copy := DryerStatus;

	//Store the history of the status to easy the debug
	IF DryerStatus<>StateHistory[0] THEN
		FOR iIndexHistory:=iHistoryLines TO 1 BY -1 DO
			StateHistory[iIndexHistory]:=StateHistory[iIndexHistory-1];
		END_FOR;
		StateHistory[0]:=DryerStatus;
		LogNewState;
	END_IF

	gDryer.St.DryerState := DryerStatus;

	gDryer.St.Out.xOnline := TRUE;
	gDryer.St.Out.xDryerPresent := TRUE;
	gDryer.St.Out.xTransportMoving := gBelt.states.xRuningBelt;
	gDryer.St.Out.xInRemote := gDryer.St.AutoLocation.xRemote;
	gDryer.St.Out.xError :=  DryerStatus = DRYERMACH_ERROR;
	gDryer.St.Out.xJamDetection := FALSE;

	ton_EmptyBelt.IN := gDryer.St.AutoLocation.xRemote AND gBelt.states.xRuningBelt AND NOT gDryerRemoteData.Parameters.xPrinterBeltRuning;
	ton_EmptyBelt.PT := T#20s;
	ton_EmptyBelt();
	gDryer.St.Out.xDrying := FALSE;
	gDryer.St.Out.xMediaPresent := FALSE;

	iReasonReadyToDry.0 := DryerStatus = DRYERMACH_PREPARED;
	iReasonReadyToDry.1 := DryerStatus = DRYERMACH_STARTING;
	iReasonReadyToDry.2 := DryerStatus = DRYERMACH_DRYING;
	gDryer.St.Out.xReadyToDry :=  iReasonReadyToDry > 0;

	gDryerLocalData.xError := gDryer.AlSummary.xAlarmCritical OR gDryer.AlSummary.xAlarmStop;
	gDryerLocalData.xDrying := DryerStatus = DRYERMACH_DRYING OR DryerStatus = DRYERMACH_STARTING;
	gDryerLocalData.xReadyToDry := gDryer.St.Out.xReadyToDry;
	gDryerLocalData.xJamDetection := gDryer.Al.Alarm.xAlrJam;
	gDryerLocalData.xTransportMoving := gBelt.states.xRuningBelt;
	gDryerLocalData.xInRemote := gDryer.St.AutoLocation.xRemote;
	gDryerLocalData.xMediaPresent := gThicknessCtrl.status.MediaPosition.xMediaBelowMachine;
	gDryerLocalData.xBeltEmpty := gThicknessCtrl.status.Belt.xBeltEmpty OR ton_EmptyBelt.Q;
	gDryerLocalData.xStopButtonPressed := gDryer.In.Buttons.xStop;
	gDryerLocalData.xReadyToEmptyBelt := gDryer.St.Out.xReadyToEmptyBelt;

	gDryer.St.Out.iModelVersion1 := gPLC.iVersion0;
	gDryer.St.Out.iModelVersion2 := gPLC.iVersion1;

END_ACTION

ACTION ResetOrdersToAllDryersDevices:
	ResetOrdersToArcLamp;
	ResetOrdersToNirAdphos;
END_ACTION

ACTION ResetOrdersToArcLamp:
	gArcLampGew.Commands.xPrepare := FALSE;
	gArcLampGew.Commands.xStart := FALSE;
	gArcLampGew.Commands.xStop := FALSE;
END_ACTION

ACTION ResetOrdersToNirAdphos:
	gNirAdphos.Commands.xPrepare := FALSE;
	gNirAdphos.Commands.xStart := FALSE;
	gNirAdphos.Commands.xStop := FALSE;
END_ACTION
```

#### EventLog.st
```iecst
ACTION LogCriticalAlarm:

	stEventLogCritical.Source := ELOG_TYPE_GENERAL;
	stEventLogCritical.Severity:= ELOG_SEVERITY_ERROR;
	stEventLogCritical.Facility:= 0;
	stEventLogCritical.ErrorCode:=0;

	stEventLogCritical.Text := 'Gen.LogCriticalAlarm';

	IF 		iReasonCritical.0 THEN stEventLogCritical.Text := 'Gen Critical. xAlrSafetySystemGeneral';
	ELSIF 	iReasonCritical.1 THEN stEventLogCritical.Text := 'Gen Critical. Belt Crical Alarm';
	ELSIF 	iReasonCritical.2 THEN stEventLogCritical.Text := 'Gen Critical. NIR Crical Alarm';
	ELSIF 	iReasonCritical.3 THEN stEventLogCritical.Text := 'Gen Critical. ARC LAMP Crical Alarm';
	ELSIF 	iReasonCritical.4 THEN stEventLogCritical.Text := 'Gen Critical. TransVacuum Crical Alarm';
	END_IF

	gEventLogLoader(EventData := ADR(stEventLogCritical));

END_ACTION

ACTION LogStopDryingAlarm:

	stEventLogStopDrying.Source := ELOG_TYPE_GENERAL;
	stEventLogStopDrying.Severity:= ELOG_SEVERITY_ERROR;
	stEventLogStopDrying.Facility:= 0;
	stEventLogStopDrying.ErrorCode:=0;

	stEventLogStopDrying.Text := 'Gen.LogStopDryingAlarm';

	IF 		iReasonStopDrying.0 THEN stEventLogStopDrying.Text := 'Gen StopDrying. xAlrBeltOvertorque';
	ELSIF 	iReasonStopDrying.1 THEN stEventLogStopDrying.Text := 'Gen StopDrying. xAlrBeltOverTempFast';
	ELSIF 	iReasonStopDrying.2 THEN stEventLogStopDrying.Text := 'Gen StopDrying. xAlrBeltOverTempSlow';
	END_IF

	gEventLogLoader(EventData := ADR(stEventLogStopDrying));

END_ACTION

ACTION LogOutOfAuto:

	stEventLogOutAuto.Source := ELOG_TYPE_GENERAL;
	stEventLogOutAuto.Severity:= ELOG_SEVERITY_INFO;
	stEventLogOutAuto.Facility:= 0;
	stEventLogOutAuto.ErrorCode:=0;

	stEventLogOutAuto.Text := 'Gen.LogOutOfAuto';

	IF 		iReasonOut.0 AND enPrinterState=PRINTERGEN_MANUAL THEN stEventLogOutAuto.Text := 'OutOfMan. Selector to Zero';
	ELSIF 	iReasonOut.0 AND enPrinterState=PRINTERGEN_AUTO THEN stEventLogOutAuto.Text := 'OutOfAuto. Selector to Zero';
	ELSIF 	iReasonOut.1 THEN stEventLogOutAuto.Text := 'OutOfAuto. Selector NOT Auto';
	ELSIF 	iReasonOut.2 THEN stEventLogOutAuto.Text := 'OutOfMan. Selector NOT Manual';
	ELSIF 	iReasonOut.3 THEN stEventLogOutAuto.Text := 'OutOfAuto. Critical Alarm';
	ELSIF 	iReasonOut.4 AND enPrinterState=PRINTERGEN_MANUAL THEN stEventLogState.Text := 'OutOfMan. Emergency alarm';
	ELSIF 	iReasonOut.4 AND enPrinterState=PRINTERGEN_AUTO THEN stEventLogOutAuto.Text := 'OutOfAuto. Emergency alarm';
	END_IF

	gEventLogLoader(EventData := ADR(stEventLogOutAuto));

END_ACTION

ACTION LogNewState:

	stEventLogState.Source := ELOG_TYPE_GENERAL;
	stEventLogState.Severity:= ELOG_SEVERITY_INFO;
	stEventLogState.Facility:= 0;
	stEventLogState.ErrorCode:=0;

	stEventLogState.Text := 'NewState. Unknown';

	CASE DryerStatus OF
		DRYERMACH_STOPPED: 				stEventLogState.Text := 'NewState. Stopped';
		DRYERMACH_STOPPING_TRANSPORT:	stEventLogState.Text := 'NewState. StoppingTransport';
		DRYERMACH_PREPARINGTOMOVE:		stEventLogState.Text := 'NewState. PreparingToMove';
		DRYERMACH_MOVING:				stEventLogState.Text := 'NewState. Moving';
		DRYERMACH_PREPARING:			stEventLogState.Text := 'NewState. Preparing';
		DRYERMACH_PREPARED:				stEventLogState.Text := 'NewState. Prepared';
		DRYERMACH_STARTING:				stEventLogState.Text := 'NewState. Starting';
		DRYERMACH_DRYING:				stEventLogState.Text := 'NewState. Drying';
		DRYERMACH_STOPPING_DRYING:		stEventLogState.Text := 'NewState. StoppinDrying';
	END_CASE;

	gEventLogLoader(EventData := ADR(stEventLogState));

END_ACTION

ACTION LogStopAlarm:

	//Alarms stop//
	stEventLog.Source := ELOG_TYPE_GENERAL;
	stEventLog.Severity:= ELOG_SEVERITY_ERROR;
	stEventLog.Facility:= 0;
	stEventLog.ErrorCode:=0;

	stEventLog.Text := 'Gen.LogStopAlarm';

	IF 		iReasonStopGen.0 THEN stEventLog.Text := 'Gen Stop. xAlarmAir1';
	ELSIF 	iReasonStopGen.1 THEN stEventLog.Text := 'Gen Stop. xAlarmComPcPLC';
	ELSIF 	iReasonStopGen.2 THEN stEventLog.Text := 'Gen Stop. xAlarmMountedMedia';
	ELSIF 	iReasonStopGen.3 THEN stEventLog.Text := 'Gen Stop. xAlrBeltOvertorque';
	ELSIF 	iReasonStopGen.4 THEN stEventLog.Text := 'Gen Stop. xAlrBeltOverTempFast';
	ELSIF 	iReasonStopGen.5 THEN stEventLog.Text := 'Gen Stop. xAlrBeltOverTempSlow';
	ELSIF 	iReasonStopGen.6 THEN stEventLog.Text := 'Gen Stop. Belt.AlarmStop';
	ELSIF 	iReasonStopGen.7 THEN stEventLog.Text := 'Gen Stop. SimpleBlock[1].xAlarmStop';
	ELSIF 	iReasonStopGen.8 THEN stEventLog.Text := 'Gen Stop. NirAdphos.AlarmStop';
	ELSIF 	iReasonStopGen.9 THEN stEventLog.Text := 'Gen Stop. ArcLampGew.AlarmStop';
	ELSIF 	iReasonStopGen.10 THEN stEventLog.Text := 'Gen Stop. gTransVacuum[1].AlarmStop';
	ELSIF 	iReasonStopGen.11 THEN stEventLog.Text := 'Gen Stop. NirAdphos.AnyJam';
	ELSIF 	iReasonStopGen.12 THEN stEventLog.Text := 'Gen Stop. ArcLampGew.Jam';
	END_IF

	gEventLogLoader(EventData := ADR(stEventLog));

END_ACTION
```

#### OrdersDryer.st
```iecst
ACTION OrdersPrinter:

	////////////////////////////////////////////////////////
	// Inputs by comns are auto commands in printer, not all
	//	from kernel: xMute_GI and xReset_GI
	//  from panel: xReset or validate
	////////////////////////////////////////////////////////

	gDryer.St.Position.xInCap := gSimpleBlock[1].Status.Position.xInCap;
	gDryer.St.Position.xInPrint := gSimpleBlock[1].Status.Position.xInPrint;
	gDryer.St.Position.xGoingToCap := gSimpleBlock[1].Status.Position.xGoingToCap;
	gDryer.St.Position.xGoingToPrint := gSimpleBlock[1].Status.Position.xGoingToPrint;
	xOrderToCapReceived	:= gSimpleBlock[1].Status.Position.xInCap OR gSimpleBlock[1].Status.Position.xGoingToCap;
	xOrderToPrintReceived := gSimpleBlock[1].Status.Position.xInPrint OR gSimpleBlock[1].Status.Position.xGoingToPrint;

	// With these bool are set enPrinterStatesInAuto
	//
	IF gDryer.St.Position.xInCap		THEN enPrinterStatesInAuto:=PRINTER_CAPPED;         END_IF
	IF gDryer.St.Position.xInPrint		THEN enPrinterStatesInAuto:=PRINTER_PRINTING;       END_IF
	IF gDryer.St.Position.xGoingToCap	THEN enPrinterStatesInAuto:=PRINTER_GOING_TO_CAP;   END_IF
	IF gDryer.St.Position.xGoingToPrint	THEN enPrinterStatesInAuto:=PRINTER_GOING_TO_PRINT; END_IF

	/////////////////////////////////////////////////////////////////////////////////
	/////////////////////////////////////////////////////////////////////////////////
	//   General auto commads to send block to print or cap from kernel			   //
	/////////////////////////////////////////////////////////////////////////////////
	/////////////////////////////////////////////////////////////////////////////////

	// An edge of commandbooledge must go to cap
	iReasonCap.0 := gDryer.commands.xAllToCap AND (NOT gDryer.St.Position.xInCap);
	iReasonCap.1 := EDGEPOS(gDryer.St.AutoMode.xStop);
	iReasonCap.2 := EDGEPOS(gDryer.St.AutoMode.xBypass);

	iReasonPrint.0 := EDGEPOS(gDryer.commands.xAllToPrint) AND (NOT gDryer.St.Position.xInPrint) AND gDryer.St.AutoMode.xProdORLab ; // An edge of commandbooledge must go to print, if the machine is not stopped
	iReasonPrint.1 := EDGEPOS (gDryer.St.AutoMode.xProduction); // An edge of auto run must go to print
	iReasonPrint.2 := gDryer.AutoCmd.xStart AND (NOT gDryer.St.Position.xInPrint) AND gDryer.St.AutoMode.xProduction; // Printer is Production, block was send to cap and then pause. It recovery to print when press play or start from gui

	IF  iReasonCap > 0 THEN

		lastReasonCap := iReasonCap;
		gDryer.AutoCmd.xToCap:= TRUE;
		gDryer.AutoCmd.xToPrint:= FALSE;
		iBlockExecutionsOrder := gSimpleBlock[1].Status.execTimes;

		// An edge of commandbooledge must go to print, if the machine is not stopped
	ELSIF iReasonPrint > 0 THEN

		lastReasonPrint := iReasonPrint;
		gDryer.AutoCmd.xToCap:= FALSE;
		gDryer.AutoCmd.xToPrint:= TRUE;
		iBlockExecutionsOrder := gSimpleBlock[1].Status.execTimes;

	END_IF

	//Fall down orders when received by the blocks
	IF EDGEPOS(xOrderToCapReceived) THEN
		gDryer.AutoCmd.xToCap := FALSE;
		iBlockDelay := gSimpleBlock[1].Status.execTimes - iBlockExecutionsOrder;
	END_IF
	IF EDGEPOS(xOrderToPrintReceived) THEN
		gDryer.AutoCmd.xToPrint := FALSE;
		iBlockDelay := gSimpleBlock[1].Status.execTimes - iBlockExecutionsOrder;
	END_IF

	//When receiving the order to go to print, update the array to avoid going down lower than needed
	IF EDGEPOS(gDryer.AutoCmd.xToPrint) OR EDGEPOS(gDryer.AutoCmd.xToCap) THEN
		gThicknessCtrl.Commands.UpdateAllMatrix:=TRUE;
	END_IF

	////////////////////////////////////////////////////////////////////////////////
	////////////////////////////////////////////////////////////////////////////////
	/////////////   THICKNESS DETECTION	THICKNESS DETECTION        /////////////////
	/////////////   THICKNESS DETECTION	THICKNESS DETECTION        /////////////////
	////////////////////////////////////////////////////////////////////////////////
	////////////////////////////////////////////////////////////////////////////////

	gThicknessCtrl.parameters.Belt.rBeltSpeed 				:= gBelt.states.rCurrentSpeed;
	gThicknessCtrl.parameters.Belt.rMinBeltSpeedToStart		:= gc_rMinSpeedToStart;
	gThicknessCtrl.parameters.ContinuousMedia.MediaData.rThickness := gDryer.Pt.SW.Media.rThickness;
	gThicknessCtrl.parameters.ContinuousMedia.MediaData.rMargin := gDryer.Pt.SW.Media.rMargin;
	gThicknessCtrl.parameters.AutoMode 	:= gDryer.St.AutoMode;

	gThicknessCtrl.parameters.Dry.rSubstratePowerReduction := gDryer.Pt.SW.rSubstratePowerReduction;

	gThicknessCtrl.Commands.xErrorRst := gDryer.AutoCmd.xReset;

	gBasicDetectMedia.Parameters.rDesiredHeigh := gDryer.Pt.SW.Media.rThickness + gDryer.Pt.SW.Media.rMargin;
	gBasicDetectMedia.Parameters.xBeltMoving := gBelt.states.xRuningBelt;
	gBasicDetectMedia.Commands.StateMode  := gDryer.St.StateMode;
	gBasicDetectMedia.Commands.AutoMode 	:= gDryer.St.AutoMode;
	gBasicDetectMedia.Commands.xReset		:= gDryer.AutoCmd.xReset;
	gBasicDetectMedia.Commands.xMute		:= gDryer.AutoCmd.xMuteAlarms;

	///////////////////////////////////////////////////////////////////////////////////
	///////////////////////////////////////////////////////////////////////////////////
	/////////////   BLOCK BLOCK BLOCK BLOCK BLOCK BLOCK BLOCK      ////////////////////
	/////////////   BLOCK BLOCK BLOCK BLOCK BLOCK BLOCK BLOCK      ////////////////////
	///////////////////////////////////////////////////////////////////////////////////
	///////////////////////////////////////////////////////////////////////////////////
	xEdgeStop := EDGEPOS(gDryer.In.Buttons.xStop);
	FOR iIndexBlock:=GC_FIRST_BLOCK TO gDryer.Pt.CT.iNumBlocks DO

		// It sends blocks to printing state because is required by mode active printer
		gSimpleBlock[iIndexBlock].commands.Mode  		:= gDryer.St.Mode;
		gSimpleBlock[iIndexBlock].commands.StateMode 	:= gDryer.St.StateMode;
		gSimpleBlock[iIndexBlock].commands.AutoMode		:= gDryer.St.AutoMode;
		gSimpleBlock[iIndexBlock].commands.xToCap		:= gDryer.AutoCmd.xToCap;
		//Avoid going arclamp to print if not enabled
		gSimpleBlock[iIndexBlock].commands.xToPrint		:= gDryer.AutoCmd.xToPrint AND gArcLampGew.Status.xEnabledArcLamp;
		gSimpleBlock[iIndexBlock].commands.xReset		:= gDryer.AutoCmd.xReset;
		gSimpleBlock[iIndexBlock].commands.xMute		:= gDryer.AutoCmd.xMuteAlarms;
		IF xEdgeStop THEN
			gSimpleBlock[iIndexBlock].commands.xBarHomeOrder := FALSE;
		END_IF

		gSimpleBlock[iIndexBlock].parameters.Motor.rPrintPosition	:= gThicknessCtrl.status.Heigh.rMaxHeigh[iIndexBlock];
		gSimpleBlock[iIndexBlock].parameters.xLeftHandMachine		:= gDryer.Pt.xLeftHandMachine;
		gSimpleBlock[iIndexBlock].parameters.xRightHandMachine		:= gDryer.Pt.xRightHandMachine;

	END_FOR

	///////////////////////////////////////////////////////////////////////////////////
	///////////////////////////////////////////////////////////////////////////////////
	/////////////   BELT  BELT  BELT  BELT  BELT  BELT  BELT  BELT  ///////////////////
	/////////////   BELT  BELT  BELT  BELT  BELT  BELT  BELT  BELT  ///////////////////
	///////////////////////////////////////////////////////////////////////////////////
	///////////////////////////////////////////////////////////////////////////////////

	//Writing belt commands
	gBelt.commands.xMute      	:= gDryer.AutoCmd.xMuteAlarms;
	gBelt.commands.xReset     	:= gDryer.AutoCmd.xReset;
	gBelt.commands.Mode 		:= gDryer.St.Mode;
	gBelt.commands.AutoMode		:= gDryer.St.AutoMode;
	gBelt.commands.xRunBelt	  	:= g_xRunBeltOrderAuto OR g_xRunBeltOrderManual;

	///////////////////////////////////////////////////////////////////////////////////
	///////////////////////////////////////////////////////////////////////////////////
	/////////////   TRANSPORT VACUUM   TRANSPORT VACUUM     ///////////////////////////
	/////////////   TRANSPORT VACUUM   TRANSPORT VACUUM     ///////////////////////////
	///////////////////////////////////////////////////////////////////////////////////
	///////////////////////////////////////////////////////////////////////////////////

	//Conditions to keep blowers running when dryer is not drying
	iReasonKeepBlowersOn.0 := gDryer.Al.Alarm.xAlrJam;
	iReasonKeepBlowersOn.1 := gBasicDetectMedia.Alarms.xMountedMedia;
	iReasonKeepBlowersOn.2 := gThicknessCtrl.status.MediaPosition.xMediaInside;
	iReasonKeepBlowersOn.3 := gThicknessCtrl.Alarms.CheckMedia[1] OR gThicknessCtrl.Alarms.CheckMedia[2];

	IF EDGENEG(gDryer.St.DryerState = DRYERMACH_DRYING) AND gDryer.St.DryerState <> DRYERMACH_STOPPING_DRYING AND iReasonKeepBlowersOn > 0 THEN
		xKeepBlowersOn := TRUE;
	ELSIF gDryer.St.DryerState  = DRYERMACH_PREPARING OR (NOT gThicknessCtrl.status.MediaPosition.xMediaInside AND NOT (gThicknessCtrl.Alarms.CheckMedia[1] OR gThicknessCtrl.Alarms.CheckMedia[2]))OR gDryer.In.Sw.xStopBlowers_GI OR gDryer.In.Buttons.xStopBlowers THEN
		xKeepBlowersOn := FALSE;
	END_IF
	gDryer.Out.xKeepSafetyNIR := xKeepBlowersOn;

	FOR usiIndex:=1 TO gDryer.Pt.CT.iNumTransVacuum BY 1 DO
		OrdersToTransVacuum;
	END_FOR

	//////////////////////////////////////////////////////////////
	//	AUTO MODE:	Order g_xRunBeltOrderAuto previous Start
	//////////////////////////////////////////////////////////////

	IF gDryer.St.Position.xCleaning AND (gDryer.St.xMediaDetected) AND NOT gDryer.St.AutoMode.xBypass THEN
		xStopBeltWhileCleaning:= TRUE;
	ELSIF NOT gDryer.St.Mode.xAuto OR NOT gDryer.St.Position.xCleaning THEN
		xStopBeltWhileCleaning:= FALSE;
	END_IF;

	xSignalsStopBeltAuto:= 	(gDryer.AlSummary.xAlarmStop AND NOT gDryer.St.AutoMode.xBypass) OR
							gDryer.Al.Alarm.xAlarmMountedMedia OR
							xStopBeltWhileCleaning;

	xAlarmsStopBeltRun:=  gDryer.AlSummary.xAlrSafetySystemGeneral;

	//Not stop de belt while the user raises the bars
	IF gDryer.commands.xAllToCap THEN
		xUserRaisesBlocks := TRUE;
	END_IF
	IF NOT gDryer.St.AutoMode.xProduction OR EDGEPOS(gDryer.St.Position.xInPrint) THEN
		xUserRaisesBlocks := FALSE;
	END_IF

	xRunBeltNormal:= gDryer.St.AutoMode.xProduction AND NOT xAlarmsStopBeltRun AND xOrdersRunBeltProduction;

	xRunBeltByPass := gDryer.St.AutoMode.xBypass; //Start bypass with run belt order. Stopped by pause when desired

	xRunBeltLab:= gDryer.St.AutoMode.xLaboratory AND NOT xAlarmsStopBeltRun;

	//Consider PAUSE just with the final order. Not in the 3 previous
	g_xRunBeltOrderAuto	:= ( xRunBeltNormal OR xRunBeltByPass OR xRunBeltLab ) AND NOT xSignalsStopBeltAuto AND NOT gDryer.St.AutoMode.xPause;

	//Printer gives consent to belt here
	gBelt.commands.xConsentBelt:=gDryer.St.xConsent OR gDryer.St.AutoMode.xLaboratory;

	///////////////////////////////////////////////////////////////////////////////////
	/////////////   ArcLamp ArcLamp ArcLamp ArcLamp ArcLamp ArcLamp ///////////////////
	/////////////   ArcLamp ArcLamp ArcLamp ArcLamp ArcLamp ArcLamp ///////////////////
	///////////////////////////////////////////////////////////////////////////////////

	gArcLampGew.Parameters.xEnableArcLamp := gDryer.Pt.SW.xEnableArcLamp;

	gArcLampGew.Parameters.StateMode := gDryer.St.StateMode;
	gArcLampGew.Parameters.AutoMode := gDryer.St.AutoMode;
	gArcLampGew.Parameters.rBeltSpeed := gBelt.states.rCurrentSpeed;
	gArcLampGew.Parameters.xBeltRunning := gBelt.states.xRuningBelt;

	gArcLampGew.Commands.xMute := gDryer.AutoCmd.xMuteAlarms;
	gArcLampGew.Commands.xReset := gDryer.AutoCmd.xReset;
	gArcLampGew.Commands.xExternalSafetyStop := gDryer.Al.Alarm.xAlrJam;
	gArcLampGew.Commands.xMediaInside := gThicknessCtrl.status.MediaPosition.xMediaInside;

	// THE COMMANDS HAVE BEEN MOVED TO THE MACHINE STATUS ITSELF

	///////////////////////////////////////////////////////////////////////////////////
	/////////////   NIR NIR NIR NIR NIR NIR NIR NIR NIR NIR NIR NIR ///////////////////
	/////////////   NIR NIR NIR NIR NIR NIR NIR NIR NIR NIR NIR NIR ///////////////////
	///////////////////////////////////////////////////////////////////////////////////

	gNirAdphos.Parameters.xEnableNir := gDryer.Pt.SW.xEnableNir;
	gNirAdphos.Parameters.DDC.xEnableDDC := gDryer.Pt.SW.xEnableDDC AND NOT gDryer.Pt.xLocalDisableDDC;

	gNirAdphos.Parameters.StateMode := gDryer.St.StateMode;
	gNirAdphos.Parameters.AutoMode := gDryer.St.AutoMode;

	//NOZDRYER-467
	IF gDryer.St.AutoLocation.xRemote AND gDryer.Pt.xEnableDryDocWidth THEN
		IF gDryer.Pt.SW.xDoubleLine THEN
			gNirAdphos.Parameters.MediaWidth := REAL_TO_INT( MIN( 	2* MAX(gDryer.Pt.SW.Media.rWidth + gDryer.Pt.SW.Media.rCrossOffset,
																			gDryer.Pt.SW.Media.rDocWidth + gDryer.Pt.SW.Media.rDocCrossOffset),
																			//gDryer.Pt.SW.Document.rWidth + gDryer.Pt.SW.Document.rOffsetL2), //There is no Line2. Big refactoring if needed
																		1400.0));
		ELSE
			gNirAdphos.Parameters.MediaWidth := REAL_TO_INT( MIN( 	2* MAX(gDryer.Pt.SW.Media.rWidth + gDryer.Pt.SW.Media.rCrossOffset,
																			gDryer.Pt.SW.Media.rDocWidth + gDryer.Pt.SW.Media.rDocCrossOffset),
																		1400.0));
		END_IF
	ELSE
		gNirAdphos.Parameters.MediaWidth := REAL_TO_INT(gDryer.Pt.SW.Media.rWidth);

	END_IF

	gNirAdphos.Parameters.rBeltSpeed := gBelt.states.rCurrentSpeed;
	gNirAdphos.Parameters.xBeltRunning := gBelt.states.xRuningBelt;
	gNirAdphos.Parameters.xLineEmptyingBelt := DryerSignalsAuto.Parameters.xLineEmptyingBelt AND gDryer.St.AutoLocation.xRemote;
	gNirAdphos.Parameters.iExtraDryingWidh := ABS(REAL_TO_INT(gThicknessCtrl.parameters.Dry.rDryExtend * 2)); // Neeed to multiply by two to consider both sides

	gNirAdphos.Commands.xMute := gDryer.AutoCmd.xMuteAlarms;
	gNirAdphos.Commands.xReset := gDryer.AutoCmd.xReset;
	gNirAdphos.Commands.xExternalSafetyStop := gDryer.Al.Alarm.xAlrJam;
	gNirAdphos.Commands.xMediaInside := gThicknessCtrl.status.MediaPosition.xMediaInside;

	gNirAdphos.Orders.xCheckJam := gBelt.states.xRuningBelt;

	IF gDryer.St.iJamDevices > 0 THEN
		//Jam
		gJamDetect[1].Commands.xReset 		:= gDryer.AutoCmd.xReset;
		gJamDetect[1].Commands.xMuteAlarms	:= gDryer.AutoCmd.xMuteAlarms;
		gJamDetect[1].Commands.xStart 		:= gDryer.St.StateMode <> PRINTERGEN_ZERO;
		gJamDetect[1].Commands.xPause		:= NOT gBelt.states.xRuningBelt;
	END_IF

	///////////////////////////////////////////////////////////////////////////////////
	//////////Cooling PC Cabinet///////////
	gDryer.Out.xCoolingPCStart := TRUE; //ALX - For the moment is On avery time, its posible control this but its necesary check in machine

	//Removing the commands
	gDryer.commands.xAllToCap:=FALSE;
	gDryer.commands.xAllToPrint:=FALSE;

END_ACTION

ACTION OrdersToTransVacuum:

	IF NOT gTransVacuum[usiIndex].Status.xInstalled THEN
		RETURN;
	END_IF

	//Avoid memory when not in manual
	IF gDryer.St.StateMode <> PRINTERGEN_MANUAL THEN
		gTransVacuum[usiIndex].OrdersSw.xRunManual := FALSE;
	END_IF

	//If needed to send parameters to other TransVacuum
	IF NOT gDryer.Pt.xTransVacuumIndependenParams AND usiIndex>1 THEN
		gTransVacuum[usiIndex].OrdersSw.xRunManual					:= gTransVacuum[1].OrdersSw.xRunManual;
		gTransVacuum[usiIndex].parSw.xActiveOutOfProduction 		:= gTransVacuum[1].parSw.xActiveOutOfProduction;
		gTransVacuum[usiIndex].parSw.rManSetPoint				:= gTransVacuum[1].parSw.rManSetPoint;
		gTransVacuum[usiIndex].Parameters.rStartUpDutyCycle			:= gTransVacuum[1].Parameters.rStartUpDutyCycle;
		gTransVacuum[usiIndex].parSw.rVacPressureSetPointPerc	:= gTransVacuum[1].parSw.rVacPressureSetPointPerc;
	END_IF

	gTransVacuum[usiIndex].Commands.xMute := gDryer.AutoCmd.xMuteAlarms;
	gTransVacuum[usiIndex].Commands.xReset := gDryer.AutoCmd.xReset;

	gTransVacuum[usiIndex].Parameters.AutoMode := gDryer.St.AutoMode;
	IF NOT xKeepBlowersOn THEN
		gTransVacuum[usiIndex].Parameters.Mode := gDryer.St.Mode;
	END_IF

	gTransVacuum[usiIndex].Commands.xRunProduction := (gBelt.states.xOrderRuning OR gThicknessCtrl.status.MediaPosition.xMediaInside OR gDryer.St.DryerState = DRYERMACH_PREPARINGEMPTYBELT) AND NOT xKeepBlowersOn;
	gTransVacuum[usiIndex].Commands.xRunMaxDutyCycle := xKeepBlowersOn;

END_ACTION
```

### Program Logical/Dryer/DryerSimAnc/DryerSimAnc_v1/DryerSimAnc

#### DryerSimAnc.var
```iecst
VAR
	SimDryer : REFERENCE TO PrimerSim_typ;
	Dryer : REFERENCE TO DryerAnc_typ;
	tonTransport : TON;
	tonReady : TON;
	tonDry : TON;
END_VAR
```

#### DryerSimAnc.st
```iecst
PROGRAM _CYCLIC
	(* Insert code here *)
	Dryer ACCESS ADR(gDryerAnc);
	SimDryer ACCESS ADR(gSimDryerAnc);

	Dryer.Inputs.xError:=SimDryer.Commands.CreateError;

	tonTransport.IN:= Dryer.Outputs.xRunTransport;
	tonTransport.PT:= T#1s;
	tonTransport();
	Dryer.Inputs.xTransportMoving:=tonTransport.Q;

	tonReady.IN:= Dryer.Inputs.xTransportMoving AND Dryer.Outputs.xPrepareToDry;
	tonReady.PT:= T#2s;
	tonReady();
	Dryer.Inputs.xReadyToDry:=tonReady.Q;

	tonDry.IN:= Dryer.Inputs.xReadyToDry AND Dryer.Outputs.xStartDrying;
	tonDry.PT:= T#1s;
	tonDry();
	Dryer.Inputs.xDrying:=tonDry.Q;

	Dryer.Inputs.xBeltEmpty:=TRUE;
	Dryer.Inputs.xCommsOK:=TRUE;
END_PROGRAM
```

### Program Logical/Dryer/HMI/HMI (IEC)

#### HMI.st - Init, cyclic, exit code
```iecst
PROGRAM _INIT

	X20AT4222_209.TempInput[1]:=123;
	X20AT4222_209.TempInput[2]:=234;
	X20AT4222_209.TempInput[3]:=456;
	X20AT4222_209.TempInput[4]:=567;

	//This is to assure raise alarms started with TRUE
	MpViewAlarms;
	Alarms;

END_PROGRAM

PROGRAM _CYCLIC

	MpViewAlarms;

	Alarms;

	IF EDGEPOS(xTest) THEN
		myValue := MpAlarmXSet(gAlrCore, 'Dryer.Alarm.BeltAnyDriveAlarm');
	ELSIF EDGENEG(xTest) THEN
		myValue := MpAlarmXReset(gAlrCore, 'Dryer.Alarm.BeltAnyDriveAlarm');
		myValueAck := MpAlarmXAcknowledge(gAlrCore, 'Dryer.Alarm.BeltAnyDriveAlarm');
	END_IF

	IF EDGEPOS(xTest2) THEN
		myValue2 := MpAlarmXSet(gAlrCore, 'Alarm2');
	ELSIF EDGENEG(xTest2) THEN
		myValue2 := MpAlarmXReset(gAlrCore, 'Alarm2');
		myValueAck2 := MpAlarmXAcknowledge(gAlrCore, 'Alarm2');
	END_IF

	xNone := MpAlarmXCheckState(gAlrCore, 'Dryer.Alarm.BeltAnyDriveAlarm', mpALARMX_STATE_NONE);
	xActive := MpAlarmXCheckState(gAlrCore, 'Dryer.Alarm.BeltAnyDriveAlarm', mpALARMX_STATE_ACTIVE);
	xInactive := MpAlarmXCheckState(gAlrCore, 'Dryer.Alarm.BeltAnyDriveAlarm', mpALARMX_STATE_INACTIVE);
	xAck := MpAlarmXCheckState(gAlrCore, 'Dryer.Alarm.BeltAnyDriveAlarm', mpALARMX_STATE_ACKNOWLEDGED);
	xUnAck := MpAlarmXCheckState(gAlrCore, 'Dryer.Alarm.BeltAnyDriveAlarm', mpALARMX_STATE_UNACKNOWLEDGED);

	gDryer.St.HMI.xDryerStopped := gDryer.St.DryerState = DRYERMACH_STOPPED;
	gDryer.St.HMI.xDryerLocalStopped := gDryer.St.DryerState = DRYERMACH_STOPPED AND gDryer.St.AutoLocation.xLocalORManual;
	gDryer.St.HMI.xShowThickness := gDryer.Pt.MachineModel = DryerType_NOZ2_NIR_ARCLAMP;
	gDryer.St.HMI.xShowEnableNIR := gDryer.St.DryerState =DRYERMACH_STOPPED AND
									gDryer.St.AutoLocation.xLocalORManual AND
									gNirAdphos.Status.xAnyModuleEnabled;

	//Simulate media in AutoLocal
	IF gDryer.St.Mode.xAuto AND gDryer.St.AutoLocation.xLocal THEN
		//Starting system
		IF EDGEPOS(gDryer.St.DryerState = DRYERMACH_DRYING) THEN
			xSimulateMedia := TRUE;
		ELSIF EDGENEG(gDryer.St.DryerState = DRYERMACH_DRYING) THEN
			xSimulateMedia := FALSE;
		END_IF
	ELSE
		xSimulateMedia := FALSE;
	END_IF
	tonSimMedia.IN := xSimulateMedia AND NOT tonSimMedia.Q;
	tonSimMedia.PT := T#500ms;
	tonSimMedia();
	IF EDGEPOS(tonSimMedia.Q) THEN
		gDryer.St.HMI.xVirtualMedia := NOT gDryer.St.HMI.xVirtualMedia;
	END_IF
	IF NOT gDryer.St.Mode.xAuto OR NOT gDryer.St.AutoLocation.xLocal THEN
		gDryer.St.HMI.xVirtualMedia := FALSE;
	END_IF

END_PROGRAM

PROGRAM _EXIT

	//Cards of the Dryer
	X20DIF371_201;
	X20DIF371_202;
	X20DIF371_203;
	X20DOF322_205;
	X20DOF322_206;
	X20AI8321_207;
	X20AO4622_208;
	X20AT4222_209;

END_PROGRAM
```
